// TwinCAT 3 PLC project Samples
// Title: TF8040 PLC-Samples
// Company: Beckhoff Automation GmbH
// Author: Beckhoff Automation
// ProjectVersion: 2.1.1.0
// Description: PLC.Samples to demontrate function volume of TF8040.
// ProgramVersion: 3.1.4023.0
// libraries:
//   Tc2_Standard, * (Beckhoff Automation GmbH)
//   Tc2_System, * (Beckhoff Automation GmbH)
//   Tc2_Utilities, * (Beckhoff Automation GmbH)
//   Tc3_BA2, * (Beckhoff Automation GmbH)
//   Tc3_BA2_Common, * (Beckhoff Automation GmbH)
//   Tc3_BACnetRev14, * (Beckhoff Automation GmbH)
//   Tc3_Module, * (Beckhoff Automation GmbH)
//   Tc3_XBA, * (Beckhoff Automation GmbH)
// project tree:
//   / PlcTask.TcTTO (not stored)
//   SAMPLES/Demo/Event/ FB_Evt_Ack.TcPOU, FB_Evt_EventClasses.TcPOU (not stored), FB_Evt_Events.TcPOU, FB_Evt_Misc.TcPOU, FB_Evt_QueryCnd.TcPOU (not stored)
//   SAMPLES/Demo/Event/Function/ F_AcknowledgeEventClass.TcPOU (not stored)
//   SAMPLES/Demo/Objects/ FB_Obj_AddParam.TcPOU, FB_Obj_General.TcPOU, FB_Obj_Misc.TcPOU, FB_Obj_Sequence.TcPOU (not stored), FB_Obj_UserDefined.TcPOU (not stored)
//   SAMPLES/Demo/Objects/Misc/ E_UDef_Mode.TcDUT (not stored), FB_UDef_BValEx.TcPOU, FB_UDef_SpVal.TcPOU, FB_UDef_SpValEx.TcPOU (not stored)
//   SAMPLES/Demo/Optional Extensions/Events/ FB_MyLocalObjectEvents.TcPOU, FB_MyProjectEvents.TcPOU (not stored)
//   SAMPLES/Demo/Optional Extensions/ MAIN_OPTEXT.TcPOU
//   SAMPLES/Demo/Other/ FB_Misc.TcPOU, FB_Texts.TcPOU (not stored)
//   SAMPLES/Demo/Plant/ FB_Plt_Init1.TcPOU (not stored), FB_Plt_Init2.TcPOU (not stored), FB_Plt_Init3.TcPOU (not stored)
//   SAMPLES/Demo/Reference/ FB_Ref_Collectors.TcPOU (not stored), FB_Ref_Groups.TcPOU (not stored)
//   SAMPLES/Demo/Reference/Publish and Subscribe/ FB_Ref_PubSub_Local.TcPOU (not stored), FB_Ref_PubSub_Remote.TcPOU
//   SAMPLES/Demo/Structure/ FB_Struct_Nested.TcPOU (not stored)
//   SAMPLES/Demo/Supplement specific/BACnet/ FB_BACnet_EvtInh.TcPOU, FB_BACnet_ObjPropRef.TcPOU (not stored), FB_BACnet_RcpList.TcPOU
//   SAMPLES/Demo/Supplement specific/BACnet/Optional Extensions/Events/ FB_BACnet_MyLocalObjectEvents.TcPOU
//   SAMPLES/Demo/Supplement specific/BACnet/Optional Extensions/ MAIN_OPTEXT_BACnet.TcPOU (not stored)
//   SAMPLES/Demo/[Helper]/FunctionBlocks/Aggregates/ FB_TimerAggregateA.TcPOU (not stored), FB_ProcAggregateB.TcPOU (not stored)
//   SAMPLES/Demo/[Helper]/FunctionBlocks/Nested/ FB_NestedView.TcPOU (not stored), FB_NestedView2.TcPOU (not stored), FB_SubNestedView.TcPOU (not stored), FB_SubSubNestedView.TcPOU
//   SAMPLES/ MAIN.TcPOU
//   SAMPLES/Templates/Standard/DUTs/Enumerations/OpMod/ E_OpMod_AC.TcDUT, E_OpMod_Binary.TcDUT (not stored), E_OpMod_ClsOpn.TcDUT (not stored), E_OpMod_Step2.TcDUT (not stored)
//   SAMPLES/Templates/Standard/GVLs/ MyECIDs.TcGVL (not stored), MyLabels.TcGVL (not stored), MyProfiles.TcGVL
//   SAMPLES/Templates/Standard/POUs/Trade/General/Building/ FB_BA_Bld01.TcPOU
//   SAMPLES/Templates/Standard/POUs/Trade/General/EventClasses/ FB_BA_EC01.TcPOU
//   SAMPLES/Templates/User-defined/Objects/ FB_UDef_Obj.TcPOU (not stored)
//   SAMPLES/Templates/User-defined/Sample Weather Station/ FB_BA_MyWeatherStation.TcPOU (not stored), FB_BA_MyWeatherStationSub.TcPOU (not stored), I_BA_MyWeatherStation.TcIO, ST_BA_MyWeatherData.TcDUT
// real-time tasks:
//   TASK PlcTask: cycle T#45ms, priority 20, ADS port 350
//   TASK Device 1 (BACnet IP)_Task_58: cycle T#40ms, priority 58, ADS port 351
//   TASK Gerät 1 (BACnet IP)_QueueTask: cycle T#2ms, priority 8, ADS port 352
// I/O:
//   DEVICE Gerät 1 (BACnet IP), AmsNetId 192.168.216.1.2.1
// variable links:
//   Samples/Samples Instance <-> Device 1 (BACnet IP)
//     PlcTask Inputs/Tc3_BACnetRev14.BACnet_Globals.DefaultAdapter.BACnet_AmsNetId <-> Inputs/AmsNetId

// ---- SAMPLES/Templates/Standard/DUTs/Enumerations/OpMod/E_OpMod_AC.TcDUT
{attribute 'qualified_only'}
TYPE E_OpMod_AC :
(
	Invalid			:= 0,
	
	eOff			:= 1,
	eOn				:= 2,
	eNightCool		:= 3,
	eDisturb		:= 4,
	eSmokeExtract	:= 5,
	eFrost			:= 6,
	eFire			:= 7,
	eCentralOff		:= 8
	
) UDINT;
END_TYPE

// ---- SAMPLES/Templates/User-defined/Sample Weather Station/ST_BA_MyWeatherData.TcDUT
TYPE ST_BA_MyWeatherData :
STRUCT
	fWeatherTemperature		: REAL;
	fHumidity				: REAL;
	fBrightness				: REAL;
	fWindSpeed				: REAL;
	fWindDirection			: REAL;
	fLatitude				: REAL;
	fLongitude				: REAL;
	
	bDisturb				: BOOL;
END_STRUCT
END_TYPE

// ---- SAMPLES/Templates/Standard/GVLs/MyProfiles.TcGVL
{attribute 'qualified_only'}
VAR_GLOBAL
	{region 'Placeholder'}
		{region 'Text'}
			txtOff						: STRING						:= 'Aus';
			txtOn						: STRING						:= 'Ein';
			txtNormal					: STRING						:= 'Normal';
			txtOffnormal				: STRING						:= 'Unnormal';
			txtAlert					: STRING						:= 'Alarm';
			txtDisturb					: STRING						:= 'Störung';
			txtExceeded					: STRING						:= 'Überschritten';
			txtMonitoring				: STRING						:= 'Überwachung';
			txtProtection				: STRING						:= 'Schutzbetrieb';
			txtEconomy					: STRING						:= 'Economy';
			txtComfort					: STRING						:= 'Comfort';
		{endregion}
		{region 'Event Transition Text'}
			trnsExceeded				: T_BA_EventTransitionText		:= [txtExceeded,			txtDisturb,			txtNormal];
			trnsMonitoring				: T_BA_EventTransitionText		:= [txtMonitoring,			txtDisturb,			txtNormal];
		{endregion}
		{region 'Multistate Text'}
			txtEnergyLevel				: T_BA_StateTextArray			:= [txtProtection,			txtEconomy,			txtComfort];
		{endregion}
	{endregion}
END_VAR
VAR_GLOBAL
	{region 'Sample Templates'}
		// A
		// B
		CmdB							: FB_BA_ProfileBEvtObj			:= (sInactiveText := txtOff,			sActiveText := txtOn,			aEventTransitionText := trnsMonitoring,							nEventClassID := 11);
		// D
		// E
		// F
		// G
		// H
		// I
		// J
		// K
		// L
		// M
		// N
		// O
		// P	
		// Q
		// R
		// S	
		// t
		// U
		// v
		// W
		// X
		// Y
		// Z
	{endregion}
	{region 'Sample Objects'}
		{region 'Analog'}
			AV_Prf						: FB_BA_ProfileAEvtObj			:= (eUnit:=E_BA_Unit.eTemperature_DegreesCelsius,						aEventTransitionText:=MyProfiles.trnsExceeded,					nEventClassID:=MyECIDs.AlmStd);
			AVOp_Prf					: FB_BA_ProfileAObj				:= (eUnit:=E_BA_Unit.eTemperature_DegreesCelsius);
			AI_Prf						: FB_BA_ProfileAEvtObj			:= (eUnit:=E_BA_Unit.eTemperature_DegreesCelsius,						aEventTransitionText:=MyProfiles.trnsExceeded,					nEventClassID:=MyECIDs.AlmStd);
			AO_Prf						: FB_BA_ProfileAEvtObj			:= (eUnit:=E_BA_Unit.eTemperature_DegreesCelsius,						aEventTransitionText:=MyProfiles.trnsExceeded,					nEventClassID:=MyECIDs.AlmStd);
		{endregion}
		{region 'Binary'}
			BV_Prf						: FB_BA_ProfileBEvtObj			:= (sInactiveText := txtOff, sActiveText := txtOn,						aEventTransitionText:=MyProfiles.trnsExceeded,					nEventClassID:=MyECIDs.AlmStd);
			BVOp_Prf					: FB_BA_ProfileBObj				:= (sInactiveText := txtOff, sActiveText := txtOn);
			BI_Prf						: FB_BA_ProfileBEvtObj			:= (sInactiveText := txtOff, sActiveText := txtOn,						aEventTransitionText:=MyProfiles.trnsExceeded,					nEventClassID:=MyECIDs.AlmStd);
			BO_Prf						: FB_BA_ProfileBEvtObj			:= (sInactiveText := txtOff, sActiveText := txtOn,						aEventTransitionText:=MyProfiles.trnsExceeded,					nEventClassID:=MyECIDs.AlmStd);
		{endregion}
		{region 'Multistate'}
			MV_Prf						: FB_BA_ProfileMEvtObj			:= (aStateText:=MyProfiles.txtEnergyLevel,								aEventTransitionText:=MyProfiles.trnsExceeded,					nEventClassID:=MyECIDs.AlmStd);	
			MVOp_Prf					: FB_BA_ProfileMObj				:= (aStateText:=MyProfiles.txtEnergyLevel);
			MI_Prf						: FB_BA_ProfileMEvtObj			:= (aStateText:=MyProfiles.txtEnergyLevel,								aEventTransitionText:=MyProfiles.trnsExceeded,					nEventClassID:=MyECIDs.AlmStd);
			MO_Prf						: FB_BA_ProfileMEvtObj			:= (aStateText:=MyProfiles.txtEnergyLevel,								aEventTransitionText:=MyProfiles.trnsExceeded,					nEventClassID:=MyECIDs.AlmStd);
		{endregion}
		{region 'Misc'}
			Loop_Prf					: FB_BA_ProfileAObj				:= (eUnit:=E_BA_Unit.eOther_Percent);
			Cal_Prf						: FB_BA_ProfileBObj				:= (sInactiveText := txtOff, sActiveText := txtOn);
			SchedA_Prf					: FB_BA_ProfileAObj				:= (eUnit:=E_BA_Unit.eOther_Percent);
			SchedB_Prf					: FB_BA_ProfileBObj				:= (sInactiveText := txtOff, sActiveText := txtOn);
			SchedM_Prf					: FB_BA_ProfileMObj				:= (aStateText:=MyProfiles.txtEnergyLevel);
			Trend_Prf					: FB_BA_ProfileBObj				:= (sInactiveText := txtOff, sActiveText := txtOn);
			EvtCls_Prf					: FB_BA_Profile;
		{endregion}
		{region 'Custom'}
			MyWthSt_Prf					: FB_BA_Profile;
		{endregion}
		{region 'Collectors'}
			Col_PrfEn					: FB_BA_ProfileBObj				:= (sInactiveText := 'Nein', sActiveText := 'Ja');
			Col_PrfValA					: FB_BA_ProfileAObj				:= (eUnit:=E_BA_Unit.eTemperature_DegreesCelsius);
		{endregion}
	{endregion}
END_VAR

// ---- SAMPLES/Templates/User-defined/Sample Weather Station/I_BA_MyWeatherStation.TcIO
INTERFACE I_BA_MyWeatherStation EXTENDS I_BA_Publisher

PROPERTY Brightness : REAL
GET
END_GET
END_PROPERTY

PROPERTY Error : BOOL
GET
END_GET
END_PROPERTY

PROPERTY Humidity : REAL
GET
END_GET
END_PROPERTY

PROPERTY Latitude : REAL
GET
END_GET
END_PROPERTY

PROPERTY Longitude : REAL
GET
END_GET
END_PROPERTY

PROPERTY Ready : BOOL
GET
END_GET
END_PROPERTY

PROPERTY WeatherTemperature : REAL
GET
END_GET
END_PROPERTY

PROPERTY WindDirection : REAL
GET
END_GET
END_PROPERTY

PROPERTY WindSpeed : REAL
GET
END_GET
END_PROPERTY

END_INTERFACE

// ---- SAMPLES/Demo/Event/FB_Evt_Ack.TcPOU
// Acknowledgement-Examples.
// > One object per demonstrated 'AlarmMode'.
// > See "FB_BA_EC01" to view decleared event classes.
// [Hint]
// > All reference-variables are implemented to ease monitoring of relevant variables.
// > show the possibility to acknowledge BA objects assigned to a specific event class.
FUNCTION_BLOCK FB_Evt_Ack EXTENDS FB_BA_View
VAR               
	{region 'General'}
		bAlm_Test						: BOOL;																						// Trigger alarm for testing.
		bAlm_AckAll						: REFERENCE TO BOOL							REF= THIS^.bAcknowledgeRm;						// Acknowledge all test objects.
		bAlm_AckMode					: POINTER TO BOOL							:= ADR(XBA_Param.eEvtMgmt_AckMode);				// Used reset mode (See parameter description for more details)
	{endregion}
		 
	{region 'Simple'}
		// Intention:					Alarm that automatically disappears.
		// State on active alarm:		- "bEvent = TRUE'
		//								- "stAckedTransitions = [FALSE,true,true]'
		// State when disappeared:		- "bEvent = false'
		//								- "stAckedTransitions = [true,true,true]'
		AlmSimple_Ack					: REFERENCE TO BOOL							REF= AlmSimple.bAcknowledgeRm;
		AlmSimple_Indicated				: BOOL;
		AlmSimple_Event					: REFERENCE TO BOOL							REF= AlmSimple.bEvent;
		AlmSimple						: FB_BA_BI_Raw := (
											iParent									:= THIS^,
											sInactiveText							:= 'Normal',
											sActiveText								:= 'Alarm',
											nEventClassID							:= MyECIDs.AlmSmpl);
	{endregion}
	{region 'Standard'}
		// Intention:					Alarm that is just indicated (by acknowledge transition) when disappeared.
		// State on active alarm:		- "bEvent = TRUE'
		//								- "stAckedTransitions = [FALSE,true,true]'
		// State when disappeared:		- "bEvent = false'
		//								- "stAckedTransitions = [FALSE,true,true]'
		// State after acknowledgement:	- "bEvent = false'
		//								- "stAckedTransitions = [true,true,true]'
		AlmStandard_Ack					: REFERENCE TO BOOL							REF= AlmStandard.bAcknowledgeRm;
		AlmStandard_Indicated			: BOOL;
		AlmStandard_Event				: REFERENCE TO BOOL							REF= AlmStandard.bEvent;
		AlmStandard						: FB_BA_BI_Raw := (
											iParent									:= THIS^,
											sInactiveText							:= 'Normal',
											sActiveText								:= 'Alarm',
											nEventClassID							:= MyECIDs.AlmStd);	
	{endregion}
	{region 'Extended'}
		// Intention:					Alarm that is indicated (by acknowledge transition) and hold when disappeared.
		//								The 'bEvent' is released when an additional reset has been triggered.
		// State on active alarm:		- "bEvent = TRUE'
		//								- "stAckedTransitions = [FALSE,true,FALSE]'
		// State when disappeared:		- "bEvent = TRUE'
		//								- "stAckedTransitions = [FALSE,true,FALSE]'
		// State after acknowledgement:	- "bEvent = TRUE'
		//								- "stAckedTransitions = [true,true,FALSE]'
		// State after reset:			- "bEvent = false'
		//								- "stAckedTransitions = [true,true,true]'
		AlmExtended_Ack					: REFERENCE TO BOOL							REF= AlmExtended.bAcknowledgeRm;
		AlmExtended_Indicated			: BOOL;
		AlmExtended_Event				: REFERENCE TO BOOL							REF= AlmExtended.bEvent;
		AlmExtended						: FB_BA_BI_Raw := (
											iParent									:= THIS^,
											sInactiveText							:= 'Normal',
											sActiveText								:= 'Alarm',
											nEventClassID							:= MyECIDs.AlmExt);	
	{endregion}	
		 
	{region 'Acknowledge event class'}	
		// Intention:					Acknowledge all objects that reference a specific event class.
		nEventClassID					: UINT										:= 0;			// Enter ID of event class to acknowledge.
	{endregion}
		 
END_VAR

SUPER^();

AlmSimple(bRawVal:=bAlm_Test);
AlmSimple_Indicated := (NOT AlmSimple.stAckedTransitions.bToOffnormal);
AlmStandard(bRawVal:=bAlm_Test);
AlmStandard_Indicated := (NOT AlmStandard.stAckedTransitions.bToOffnormal);
AlmExtended(bRawVal:=bAlm_Test);
AlmExtended_Indicated := (NOT AlmExtended.stAckedTransitions.bToOffnormal);

IF (nEventClassID <> 0) THEN
	F_AcknowledgeEventClass(nEventClassID);
	nEventClassID := 0;
END_IF

// Intention:			Illustrate how to recognize changed events.
METHOD PROTECTED OnObjectEventChange
VAR_INPUT
	iObject				: I_BA_EventObject;
	bNotifyParents		: BOOL				:= TRUE;
END_VAR
SUPER^.OnObjectEventChange(iObject, bNotifyParents);

// Sample 1) Evaluate current event state:
CASE (iObject.EventIcon.eState) OF
	E_BA_EventIconState.eGoneAcked,
	E_BA_EventIconState.ePresentAcked:
		iObject.LogMsg.Show(ADSLOG_MSGTYPE_HINT, 'OOEC06', 'Object acknowledged.', TRUE);
END_CASE

// Sample 2) Compare actual event state to previous event state:
IF (iObject.LastEventIcon.eState < iObject.EventIcon.eState) THEN
	; // State intensed...
ELSE
	; // State softened...
END_IF
END_METHOD

END_FUNCTION_BLOCK

// ---- SAMPLES/Demo/Event/FB_Evt_Events.TcPOU
// Examples of objects that refer different event classes.
// > One object per 'EventType' and 'AlarmMode'.
// > One "PlantLock" per 'EventType'.
// > One "PlantLock" for entire view.
// > See "FB_BA_EC01" to view decleared event classes.
// [Hint]
// > All reference-variables are implemented to ease monitoring of relevant variables.
FUNCTION_BLOCK FB_Evt_Events EXTENDS FB_BA_View
VAR
	{region 'General'}
		Lock					: FB_BA_PlantLock				:= (iParent:=THIS^);
	{endregion}
		 
	{region 'Alarm'}
		Alm						: FB_BA_View					:= (iParent:=THIS^,	sDescription:='{Alarm}');
			AlmLock				: FB_BA_PlantLock				:= (iParent:=Alm);
							
			BIAlmSmpl_Val		: REFERENCE TO BOOL				REF= BIAlmSmpl.bVal;
			BIAlmSmpl_LockPrio	: POINTER TO E_BA_LockPriority	:= ADR(BIAlmSmpl.eEnPlantLock);
			BIAlmSmpl			: FB_BA_BI						:= (iParent:=Alm,	iLabel:=MyLabels.Cmd,	iProfile:=MyProfiles.CmdB,	nEventClassID:=MyECIDs.AlmSmpl);
			BIAlmStd_Val		: REFERENCE TO BOOL				REF= BIAlmStd.bVal;
			BIAlmStd_LockPrio	: POINTER TO E_BA_LockPriority	:= ADR(BIAlmStd.eEnPlantLock);
			BIAlmStd			: FB_BA_BI						:= (iParent:=Alm,	iLabel:=MyLabels.Cmd,	iProfile:=MyProfiles.CmdB,	nEventClassID:=MyECIDs.AlmStd,	eEnPlantLock:= E_BA_LockPriority.eHigh);
			BIAlmExt_Val		: REFERENCE TO BOOL				REF= BIAlmExt.bVal;
			BIAlmExt_LockPrio	: POINTER TO E_BA_LockPriority	:= ADR(BIAlmExt.eEnPlantLock);
			BIAlmExt			: FB_BA_BI						:= (iParent:=Alm,	iLabel:=MyLabels.Cmd,	iProfile:=MyProfiles.CmdB,	nEventClassID:=MyECIDs.AlmExt);
	{endregion}
	{region 'Disturb'}
		Dstb					: FB_BA_View					:= (iParent:=THIS^,	sDescription:='{Disturb}');
			DstbLock			: FB_BA_PlantLock				:= (iParent:=Dstb);

			BIDstbSmpl_Val		: REFERENCE TO BOOL				REF= BIDstbSmpl.bVal;
			BIDstbSmpl_LockPrio	: POINTER TO E_BA_LockPriority	:= ADR(BIDstbSmpl.eEnPlantLock);
			BIDstbSmpl			: FB_BA_BI						:= (iParent:=Dstb,	iLabel:=MyLabels.Cmd,	iProfile:=MyProfiles.CmdB,	nEventClassID:=MyECIDs.DstSmpl);
			BIDstbStd_Val		: REFERENCE TO BOOL				REF= BIDstbStd.bVal;
			BIDstbStd_LockPrio	: POINTER TO E_BA_LockPriority	:= ADR(BIDstbStd.eEnPlantLock);
			BIDstbStd			: FB_BA_BI						:= (iParent:=Dstb,	iLabel:=MyLabels.Cmd,	iProfile:=MyProfiles.CmdB,	nEventClassID:=MyECIDs.DstStd,	eEnPlantLock:= E_BA_LockPriority.eMedium);
			BIDstbExt_Val		: REFERENCE TO BOOL				REF= BIDstbExt.bVal;
			BIDstbExt_LockPrio	: POINTER TO E_BA_LockPriority	:= ADR(BIDstbExt.eEnPlantLock);
			BIDstbExt			: FB_BA_BI						:= (iParent:=Dstb,	iLabel:=MyLabels.Cmd,	iProfile:=MyProfiles.CmdB,	nEventClassID:=MyECIDs.DstExt);
	{endregion}
	{region 'Maintenance'}
		Mntn					: FB_BA_View					:= (iParent:=THIS^,	sDescription:='{Maintenance}');
			MntnLock			: FB_BA_PlantLock				:= (iParent:=Mntn);

			BIMntnSmpl_Val		: REFERENCE TO BOOL				REF= BIMntnSmpl.bVal;
			BIMntnSmpl_LockPrio	: POINTER TO E_BA_LockPriority	:= ADR(BIMntnSmpl.eEnPlantLock);
			BIMntnSmpl			: FB_BA_BI						:= (iParent:=Mntn,	iLabel:=MyLabels.Cmd,	iProfile:=MyProfiles.CmdB,	nEventClassID:=MyECIDs.MntnSmpl);
			BIMntnStd_Val		: REFERENCE TO BOOL				REF= BIMntnStd.bVal;
			BIMntnStd_LockPrio	: POINTER TO E_BA_LockPriority	:= ADR(BIMntnStd.eEnPlantLock);
			BIMntnStd			: FB_BA_BI						:= (iParent:=Mntn,	iLabel:=MyLabels.Cmd,	iProfile:=MyProfiles.CmdB,	nEventClassID:=MyECIDs.MntnStd,	eEnPlantLock:= E_BA_LockPriority.eLocalHigh);
			BIMntnExt_Val		: REFERENCE TO BOOL				REF= BIMntnExt.bVal;
			BIMntnExt_LockPrio	: POINTER TO E_BA_LockPriority	:= ADR(BIMntnExt.eEnPlantLock);
			BIMntnExt			: FB_BA_BI						:= (iParent:=Mntn,	iLabel:=MyLabels.Cmd,	iProfile:=MyProfiles.CmdB,	nEventClassID:=MyECIDs.MntnExt);
	{endregion}
	{region 'Notification'}
		Ntfy					: FB_BA_View					:= (iParent:=THIS^,	sDescription:='{Notification}');
			NtfyLock			: FB_BA_PlantLock				:= (iParent:=Ntfy);

			BINtfySmpl_Val		: REFERENCE TO BOOL				REF= BINtfySmpl.bVal;
			BINtfySmpl_LockPrio	: POINTER TO E_BA_LockPriority	:= ADR(BINtfySmpl.eEnPlantLock);
			BINtfySmpl			: FB_BA_BI						:= (iParent:=Ntfy,	iLabel:=MyLabels.Cmd,	iProfile:=MyProfiles.CmdB,	nEventClassID:=MyECIDs.NtfSmpl);
			BINtfyStd_Val		: REFERENCE TO BOOL				REF= BINtfyStd.bVal;
			BINtfyStd_LockPrio	: POINTER TO E_BA_LockPriority	:= ADR(BINtfyStd.eEnPlantLock);
			BINtfyStd			: FB_BA_BI						:= (iParent:=Ntfy,	iLabel:=MyLabels.Cmd,	iProfile:=MyProfiles.CmdB,	nEventClassID:=MyECIDs.NtfStd,	eEnPlantLock:= E_BA_LockPriority.eLocalMedium);
	{endregion}
	{region 'Other'}
		Other					: FB_BA_View					:= (iParent:=THIS^,	sDescription:='{Other}');
			OtherLock			: FB_BA_PlantLock				:= (iParent:=Other);
				 
			BIOthrSmpl_Val		: REFERENCE TO BOOL				REF= BIOthrSmpl.bVal;
			BIOthrSmpl_LockPrio	: POINTER TO E_BA_LockPriority	:= ADR(BIOthrSmpl.eEnPlantLock);
			BIOthrSmpl			: FB_BA_BI						:= (iParent:=Other,	iLabel:=MyLabels.Cmd,	iProfile:=MyProfiles.CmdB,	nEventClassID:=MyECIDs.OthSmpl);
			BIOthrStd_Val		: REFERENCE TO BOOL				REF= BIOthrStd.bVal;
			BIOthrStd_LockPrio	: POINTER TO E_BA_LockPriority	:= ADR(BIOthrStd.eEnPlantLock);
			BIOthrStd			: FB_BA_BI						:= (iParent:=Other,	iLabel:=MyLabels.Cmd,	iProfile:=MyProfiles.CmdB,	nEventClassID:=MyECIDs.OthStd);
	{endregion}                                                
END_VAR

SUPER^(); // FB_BA_View
Lock(); // FB_BA_PlantLock
Alm(); // FB_BA_View
AlmLock(); // FB_BA_PlantLock
BIAlmSmpl(); // FB_BA_BI
BIAlmStd(); // FB_BA_BI
BIAlmExt(); // FB_BA_BI
Dstb(); // FB_BA_View
DstbLock(); // FB_BA_PlantLock
BIDstbSmpl(); // FB_BA_BI
BIDstbStd(); // FB_BA_BI
BIDstbExt(); // FB_BA_BI
Mntn(); // FB_BA_View
MntnLock(); // FB_BA_PlantLock
BIMntnSmpl(); // FB_BA_BI
BIMntnStd(); // FB_BA_BI
BIMntnExt(); // FB_BA_BI
Ntfy(); // FB_BA_View
NtfyLock(); // FB_BA_PlantLock
BINtfySmpl(); // FB_BA_BI
BINtfyStd(); // FB_BA_BI
Other(); // FB_BA_View
OtherLock(); // FB_BA_PlantLock
BIOthrSmpl(); // FB_BA_BI
BIOthrStd(); // FB_BA_BI

END_FUNCTION_BLOCK

// ---- SAMPLES/Demo/Event/FB_Evt_Misc.TcPOU
FUNCTION_BLOCK FB_Evt_Misc EXTENDS FB_BA_View
VAR
	{region 'Iteration'}
		// Intention:			Iterate over active events.
		bIterate				: BOOL;
		bIterate_ShowTimestamp	: BOOL				:= FALSE;
		bIterate_ShowType		: BOOL				:= TRUE;
		bIterate_ShowState		: BOOL				:= TRUE;
		bIterate_ShowEC			: BOOL				:= FALSE;
	{endregion}
END_VAR
VAR
	_i							: DINT;
	_sVal						: T_MaxString;
	_iObj						: I_BA_EventObject;
	_fbMsg						: FB_BA_DecorString;
END_VAR

SUPER^();

IF (bIterate) THEN
	bIterate := FALSE;
	
	_i := F_BA_GetEventCount();
	IF (_i = 0) THEN
		F_BA_LogMessage(ADSLOG_MSGTYPE_HINT, 'EM06', 'No active events found yet.');
	ELSE
		F_BA_LogMessage1(ADSLOG_MSGTYPE_HINT, 'EM08', 'Active events: %d', F_DINT(_i));
		
		// Iterate over all active events:
		_i := 0;
		_iObj := 0;								// [Hint] Temporary iterator-object must be NULL to start iteration from the beginning.
		WHILE (F_BA_IterateEvents(_iObj)) DO
			_i := (_i+1);
			
			// Format message:
			_fbMsg.Reset();
			IF (bIterate_ShowTimestamp) THEN
				_sVal := TO_STRING(F_BA_ToDT(_iObj.EventChangeTime));
				_fbMsg.AddDecor1('%s', F_STRING(_sVal));
			END_IF
			IF (bIterate_ShowType) THEN
				_fbMsg.AddDecor1('Type: %s', F_STRINGEx(BA_EnumEN.aEventType[_iObj.EventIcon.eEventType].sName));
			END_IF
			IF (bIterate_ShowState) THEN
				_fbMsg.AddDecor1('State: %s', F_STRINGEx(BA_EnumEN.aEventIconState[_iObj.EventIcon.eState].sDescription));
			END_IF
			IF (bIterate_ShowEC) THEN
				_sVal := TO_STRING(_iObj.EventClassID);
				_fbMsg.AddDecor1('Event class: %s', F_STRING(_sVal));
			END_IF
			_fbMsg.Finish();
			
			_sVal := _iObj.ObjectName;
			F_BA_LogMessage3(ADSLOG_MSGTYPE_HINT, 'EM32', '%d. %s   %s', F_DINT(_i), F_STRING(_sVal), F_STRING(_fbMsg.sOutput));
		END_WHILE
	END_IF
END_IF

END_FUNCTION_BLOCK

// ---- SAMPLES/Demo/Objects/FB_Obj_AddParam.TcPOU
FUNCTION_BLOCK FB_Obj_AddParam EXTENDS FB_BA_View
VAR
	TestSpVal			: FB_UDef_SpVal := (
							iParent					:= THIS^,		
							sDescription			:= 'My user defined setpoint object',
							eMode					:= E_UDef_Mode.eAdd
						);
	TestSpValEx			: FB_UDef_SpValEx := (
							iParent					:= THIS^,
							sDescription			:= 'Another user defined enabled setpoint object',
							eMode					:= E_UDef_Mode.eSubstract
						);
	TestBValEx			: FB_UDef_BValEx := (
							iParent					:= THIS^,
							sDescription			:= 'My user defined boolean value extension',
							sActiveText				:= 'Active',
							sInactiveText			:= 'Inactive'
						);
END_VAR
VAR
	{region 'Test'}
		nOffset			: UINT						:= 3;
	{endregion}
END_VAR

SUPER^(); // FB_BA_View
TestSpVal(nSomeOffset := nOffset); // FB_UDef_SpVal
TestSpValEx(nSomeOffset := nOffset); // FB_UDef_SpValEx
TestBValEx(); // FB_UDef_BValEx

END_FUNCTION_BLOCK

// ---- SAMPLES/Demo/Objects/Misc/FB_UDef_SpVal.TcPOU
// User defined setpoint providing value.
// > Contains additional parameters.
FUNCTION_BLOCK FB_UDef_SpVal EXTENDS FB_BA_Object
VAR_INPUT CONSTANT
	{region 'Variable Parameters'}
		{attribute 'BaParam.Title.DE' := 'Irgendein Sollwert'}
		{attribute 'BaParam.Title.EN' := 'Some setpoint'}
		{attribute 'BaParam.Access.Read' := 'Guest'}
		{attribute 'BaParam.Access.Write' := 'Basic'}
		fSomeSetpoint : REAL := 10.0;
	{endregion}
END_VAR
VAR_INPUT
	{attribute 'BaParam.Title.DE' := 'Irgendein Offset'}
	{attribute 'BaParam.Title.EN' := 'Some offset'}
	{attribute 'BaParam.Access.Read' := 'Guest'}
	nSomeOffset : UINT := 3;
END_VAR
VAR_OUTPUT
	{attribute 'BaParam.Title.DE' := 'Ergebnis'}
	{attribute 'BaParam.Title.EN' := 'Result'}
	{attribute 'BaParam.Access.Read' := 'Guest'}
	fResult : REAL;
END_VAR
VAR
	{attribute 'BaParam.Title.DE' := 'Modus'}
	{attribute 'BaParam.Title.EN' := 'Mode'}
	{attribute 'BaParam.Access.Read' := 'Advanced'}
	{attribute 'BaParam.Access.Write' := 'Expert'}
	eMode : E_UDef_Mode := E_UDef_Mode.eAdd;
END_VAR

SUPER^();

CASE (eMode) OF
	E_UDef_Mode.eAdd: fResult := (fSomeSetpoint + TO_REAL(nSomeOffset));
	E_UDef_Mode.eSubstract: fResult := (fSomeSetpoint - TO_REAL(nSomeOffset));
ELSE
	fResult := fSomeSetpoint;
END_CASE

END_FUNCTION_BLOCK

// ---- SAMPLES/Demo/Objects/Misc/FB_UDef_BValEx.TcPOU
// User defined boolean value extension.
// > Contains additional parameters.
FUNCTION_BLOCK FB_UDef_BValEx EXTENDS FB_BA_BV_OP
VAR_INPUT CONSTANT
	{region 'Variable Parameters'}
		{attribute 'BaParam.Title.DE' := 'Erwarteter Wert'}
		{attribute 'BaParam.Title.EN' := 'Expected value'}
		{attribute 'BaParam.Access.Read' := 'Guest'}
		{attribute 'BaParam.Access.Write' := 'Advanced'}
		bExpected : BOOL;
	{endregion}
END_VAR
VAR_OUTPUT
	{attribute 'BaParam.Title.DE' := 'Übereinstimmend'}
	{attribute 'BaParam.Title.EN' := 'Matched'}
	{attribute 'BaParam.Access.Read' := 'Guest'}
	bMatch : BOOL;
END_VAR

SUPER^();

bMatch := (bPresentValue = bExpected);

END_FUNCTION_BLOCK

// ---- SAMPLES/Demo/Optional Extensions/Events/FB_MyLocalObjectEvents.TcPOU
FUNCTION_BLOCK FB_MyLocalObjectEvents EXTENDS FB_BA_LocalObjectEventSubscriber

METHOD PRIVATE IsPressure : BOOL
VAR_INPUT
	eUnit		: E_BA_Unit;
END_VAR
IsPressure := (E_BA_Unit.ePressure_Pascals <= eUnit) AND_THEN (eUnit <= E_BA_Unit.ePressure_InchesOfMercury);
END_METHOD

METHOD PRIVATE IsTemperature : BOOL
VAR_INPUT
	eUnit		: E_BA_Unit;
END_VAR
IsTemperature := (E_BA_Unit.eTemperature_DegreesCelsius <= eUnit) AND_THEN (eUnit <= E_BA_Unit.eTemperature_DegreeDaysFahrenheit);
END_METHOD

METHOD PROTECTED OnInitInstanceId
VAR_INPUT
	iObject			: I_BA_Object;
END_VAR
VAR_INST
	_nID_Temp		: UDINT						:= 5000;				// First ID to assign to temperature sensors.
	_nID_Prs		: UDINT						:= 6000;				// First ID to assign to pressure sensors.
END_VAR
VAR
	_iAnalogObj		: I_BA_AnalogObject;
	_nID			: REFERENCE TO UDINT;
END_VAR
// Sample 1) Generate instance ID related to configured units.

IF (iObject.InstanceID <> 0) THEN
	; // ID already assigned.
ELSIF (iObject.DataClass <> E_BA_DataClass.eAnalog) THEN
	; // Skip.
ELSIF (NOT __QUERYINTERFACE(iObject, _iAnalogObj)) THEN
	; // Failed to convert interface.
ELSE
	// Determine range of instance IDs:
	IF (IsTemperature(_iAnalogObj.Unit)) THEN
		_nID REF= _nID_Temp;
	ELSIF (IsPressure(_iAnalogObj.Unit)) THEN
		_nID REF= _nID_Prs;
	ELSE
		RETURN; // Skip (Instance ID will be auto-generated).
	END_IF
		
	// Assign instance ID:
	_iAnalogObj.InstanceID := _nID;
	iObject.LogMsg.Show1(ADSLOG_MSGTYPE_HINT, 'OIII21', 'Assigned instance ID %d.', F_UDINT(_nID), FALSE);
	
	_nID := (_nID+1);
END_IF
END_METHOD

END_FUNCTION_BLOCK

// ---- SAMPLES/Demo/Optional Extensions/MAIN_OPTEXT.TcPOU
// Optional extensions.
// [Hint]
// - To stay maintainable and sustain a nice project overview it is recommended to declare these tools in your MAIN program.
PROGRAM MAIN_OPTEXT
VAR
	{region 'Settings'}
		// Intention:		Adjust certain ("BA_Param" related) settings via PLC code.
		//					> Feel free to implement as much instances as needed, where ever needed.
		Parameters			: FB_BA_Param := (
								EventEn_Simple			:= F_BA_EventTransition(TRUE, FALSE, FALSE),
								EventEn_Standard		:= F_BA_EventTransition(TRUE, FALSE, FALSE),
								EventEn_Extended		:= F_BA_EventTransition(TRUE, FALSE, TRUE),
								EvtMgmt_AckMode			:= E_BA_AcknowledgeMode.eSingle,
								
								// Intention:			Adjust access to some specific parameters (Leaving rest untouched).
								DefWriteAccess			:= F_BA_ParameterRolesBuilder()
															.Set(E_BA_Parameter.eEventEnable, E_BA_Role.eInternal)
															.Build()
							);

		// Intention:		Generically subscribe to certain events.
		//					> Use carefully (Refer to documentation - event subscribers are powerfull!)
		Events_Proj			: FB_MyProjectEvents;
		Events_LocObj		: FB_MyLocalObjectEvents;
	{endregion}
END_VAR

END_PROGRAM

// ---- SAMPLES/Demo/Other/FB_Misc.TcPOU
// Miscellaneous.
FUNCTION_BLOCK FB_Misc EXTENDS FB_BA_View
VAR	
	// Intention:		Take care of UTF-8 encoding manually.
	//					> [Hint] Disable the integrated encoding mechanism (See "BA_Param.bUtf8AutoConvert")!
	SpecialUtf8			: FB_BA_AV_Op := (
							iParent					:= THIS^,
							sDescription			:= wsLiteral_TO_UTF8("{äöüßéèêµ€° Ἀθῆναι İstanbul Київ}"),
							eUnit					:= E_BA_Unit.eOther_Percent,
							fValueRm				:= 5
						);
END_VAR

SUPER^();

SpecialUtf8();

END_FUNCTION_BLOCK

// ---- SAMPLES/Demo/Objects/FB_Obj_General.TcPOU
// Demonstration of objects.
// > See "FB_BA_EC01" to view decleared event classes.
FUNCTION_BLOCK FB_Obj_General EXTENDS FB_BA_View
VAR
	{region 'Analog'}
		A										: FB_BA_View := (
													iParent									:= THIS^,
													sDescription							:= '{Analog objects}'
												);
			 
			// Intention:						Value
			AV									: FB_BA_AV := (
													iParent									:= A,
													sDescription							:= '{Analog Value}',
													eUnit									:= E_BA_Unit.eOther_Percent,
													nEventClassID							:= MyECIDs.AlmStd,
													stLowLimit								:= F_BA_Limit(TRUE, 0),
													stHighLimit								:= F_BA_Limit(TRUE, 50),
													stTimeDelay								:= F_BA_TimeDelay(1, 1),
													bEnPgm									:= TRUE,
													fValPgm									:= 10.0
												);
													
			// Intention:						Value for Display
			// Operation:						Display
			fAVDsp_ValuePgm						: REAL := 0;
			AVDsp								: FB_BA_AV_Op := (
													iParent									:= A,
													sObjectName								:= '{MyAvDsp}',
													sDescription							:= '{Sample AV Display}',
													eUnit									:= E_BA_Unit.eOther_Percent
												);	
			
			// Intention:						Value for Setpoint
			// Operation:						Setpoint
			AVSp								: FB_BA_AV_Op := (
													iParent									:= A,
													sDescription							:= '{Sample AV Setpoint}',
													eUnit									:= E_BA_Unit.eTemperature_DegreesCelsius,
													fValueRm								:= 3
												);
			bAVSp2_ValViaProp					: BOOL;
			fAVSp2_ValViaProp					: REAL;
			AVSp2								: FB_BA_AV_Op := (
													iParent									:= A,
													sDescription							:= '{Sample AV Setpoint 2}',
													eUnit									:= E_BA_Unit.eTemperature_DegreesCelsius,
													fValueRm								:= 3
												);
		
			// Intention:						Input
			// Hardware:						Process Data
			fAI_Proc_ValuePgm					: REAL := 20;
			AI_Proc								: FB_BA_AI := (
													iParent									:= A,
													sDescription							:= '{Sample AI (Process Data)}',
													sDeviceType								:= 'Analoger Eingang',
													eUnit									:= E_BA_Unit.eOther_Percent,
													nEventClassID							:= MyECIDs.AlmStd
												);
		
			// Intention:						Input
			// Hardware:						Raw Data
			AI_Raw								: FB_BA_AI_Raw := (
													iParent									:= A,
													sDescription							:= '{Sample AI (Raw)}',
													sDeviceType								:= 'Analoger Eingang',
													eUnit									:= E_BA_Unit.eOther_Percent,
													nEventClassID							:= MyECIDs.AlmStd
												);
		
			// Intention:						Input
			// Hardware:						I/O
			AI_IO								: FB_BA_AI_IO := (
													iParent									:= A,
													sDescription							:= '{Sample AI (IO)}',
													sDeviceType								:= 'Analoger Eingang',
													eUnit									:= E_BA_Unit.eOther_Percent,
													nEventClassID							:= MyECIDs.AlmStd
												);
												
			AI_IO_2_10V							: FB_BA_AI_IO := (
													iParent									:= A,
													sDescription							:= '{Sample AI (IO)}',
													sDeviceType								:= 'Analoger Eingang (2-10V)',
													eUnit									:= E_BA_Unit.eOther_Percent,
													nEventClassID							:= MyECIDs.AlmStd
												);
		
			// Intention:						Input
			// Hardware:						I/O
			AI_Temp								: FB_BA_AI_IOEx := (
													iParent									:= A,
													sDescription							:= '{Sample AI Temperaturfühler (Temp)}',
													sDeviceType								:= 'Temperaturfühler',
													eUnit									:= E_BA_Unit.eTemperature_DegreesCelsius,
													eSensor									:= E_BA_MeasuringElement.eNI1000,
													nEventClassID							:= MyECIDs.AlmStd
												);
		
			// Intention:						Input for Display
			// Operation:						Display
			// Hardware:						I/O
			// Parameter:						EventDetectionEnable = FALSE
			AIDsp_IO							: FB_BA_AI_IO := (
													iParent									:= A,
													sDescription							:= '{Sample AI Display (IO)}',
													sDeviceType								:= 'Analoger Eingang',
													eUnit									:= E_BA_Unit.eOther_Percent,
													bEventDetectionEnable					:= FALSE,
													nEventClassID							:= MyECIDs.AlmStd
												);
		
			// Intention:						Output
			// Hardware:						Process Data
			AO_CmdProc							: FB_BA_AO := (
													iParent									:= A,
													sDescription							:= '{Analog Befehl (Process Data)}',
													eUnit									:= E_BA_Unit.eOther_Percent,
													nEventClassID							:= MyECIDs.AlmStd
												);
		
			// Intention:						Output
			// Hardware:						Raw Data
			AO_CmdRaw							: FB_BA_AO_Raw := (
													iParent									:= A,
													sDescription							:= '{Analog Befehl (Raw Data)}',
													eUnit									:= E_BA_Unit.eOther_Percent,
													nEventClassID							:= MyECIDs.AlmStd
												);
		
			// Intention:						Output
			// Hardware:						I/O
			AO_CmdIO							: FB_BA_AO_IO := (
													iParent									:= A,
													sDescription							:= '{Analog Befehl (IO)}',
													eUnit									:= E_BA_Unit.eOther_Percent,
													nEventClassID							:= MyECIDs.AlmStd
												);
		
			// Intention:						Output for Display
			// Operation:						Display
			// Hardware:						I/O
			// Parameter:						EventDetectionEnable = FALSE
			AODisp_CmdIO						: FB_BA_AO_IO := (
													iParent									:= A,
													sDescription							:= '{Analog Befehl Display (IO)}',
													eUnit									:= E_BA_Unit.eOther_Percent,
													bEventDetectionEnable					:= FALSE,
													nEventClassID							:= MyECIDs.AlmStd
												);
	{endregion}
	{region 'Binary'}
		B										: FB_BA_View := (
													iParent									:= THIS^,
													sDescription							:= '{Binary objects}'
												);
			 
			// Intention:						Value
			BV									: FB_BA_BV := (
													iParent									:= B,
													sDescription							:= '{Binary Value}',
													sInactiveText							:= 'Aus',
													sActiveText								:= 'Ein',
													nEventClassID							:= MyECIDs.AlmExt
												);
															
			// Intention:						Value for Display
			// Operation:						Display
			bBVDsp_ValuePgm						: BOOL := FALSE;
			BVDsp								: FB_BA_BV_Op := (
													iParent									:= B,
													sDescription							:= '{Sample BV Display}',
													sInactiveText							:= 'Aus',
													sActiveText								:= 'Ein'
												);
			
			// Intention:						Value for Setpoint
			// Operation:						Setpoint
			BVSp								: FB_BA_BV_Op := (
													iParent									:= B,
													sDescription							:= '{Sample BV Setpoint}',
													sInactiveText							:= 'Aus',
													sActiveText								:= 'Ein',
													bValueRm								:= TRUE
												);
												
			// Intention:						Value for Setpoint
			// Operation:						Pushbutton
			nBVPushButton_Counter				: UINT;
			BVPushButton						: FB_BA_BV_Op := (
													iParent									:= B,
													sDescription							:= '{Sample BV Pushbutton}',
													sInactiveText							:= 'Aus',
													sActiveText								:= 'Ein',
													eToggleMode								:= E_BA_ToggleMode.ePushButton
												);
		
			// Intention:						Input
			// Hardware:						Process Data
			BI_Proc								: FB_BA_BI := (
													iParent									:= B,
													sDescription							:= '{Sample BI (Process Data)}',
													sDeviceType								:= 'Sicherung',
													sInactiveText							:= 'Normal',
													sActiveText								:= 'Ausgelöst',
													nEventClassID							:= MyECIDs.AlmStd
												);
		
			// Intention:						Input
			// Hardware:						Raw Data
			BI_Raw								: FB_BA_BI_Raw := (
													iParent									:= B,
													sDescription							:= '{Sample BI (Raw Data)}',
													sDeviceType								:= 'Sicherung',
													sInactiveText							:= 'Normal',
													sActiveText								:= 'Ausgelöst',
													nEventClassID							:= MyECIDs.AlmStd
												);
		
			// Intention:						Input
			// Hardware:						I/O
			BI_DstbIO							: FB_BA_BI_IO := (
													iParent									:= B,
													sDescription							:= '{Sample BI Disturb (IO)}',
													sDeviceType								:= 'Sicherung',
													sInactiveText							:= 'Normal',
													sActiveText								:= 'Ausgelöst',
													ePolarity								:= E_BA_Polarity.eReverse,
													nEventClassID							:= MyECIDs.DstStd,
													eEnPlantLock							:= E_BA_LockPriority.eLocalMedium
												);
		
			// Intention:						Input for Display
			// Operation:						Display
			// Hardware:						I/O
			// Parameter:						EventDetectionEnable = FALSE
			BIDsp_SwiIO							: FB_BA_BI_IO := (
													iParent									:= B,
													sDescription							:= '{Sample BI Schalter Display (IO)}',
													sDeviceType								:= 'Sicherung',
													sInactiveText							:= 'Normal',
													sActiveText								:= 'Ausgelöst',
													ePolarity								:= E_BA_Polarity.eReverse,
													nEventClassID							:= MyECIDs.OthSmpl,
													bEventDetectionEnable					:= FALSE
												);
		
			// Intention:						Output
			// Hardware:						I/O
			BO_CmdIO							: FB_BA_BO_IO := (
													iParent									:= B,
													sDescription							:= '{Sample BO Befehl (IO)}',
													sInactiveText							:= 'Aus',
													sActiveText								:= 'Ein',
													nEventClassID							:= MyECIDs.AlmStd,
													stTimeDelay := (
														nToAbnormal							:= 3
													)
												);
		
			// Intention:						Output
			// Hardware:						Process Data
			BO_CmdProc							: FB_BA_BO := (
													iParent									:= B,
													sDescription							:= '{Sample BO Befehl (Process Data)}',
													sInactiveText							:= 'Aus',
													sActiveText								:= 'Ein',
													nEventClassID							:= MyECIDs.AlmStd,
													stTimeDelay := (
														nToAbnormal							:= 3
													)
												);
		
			// Intention:						Output
			// Hardware:						Raw Data
			BO_CmdRaw							: FB_BA_BO_Raw := (
													iParent									:= B,
													sDescription							:= '{Sample BO Befehl (Raw Data)}',
													sInactiveText							:= 'Aus',
													sActiveText								:= 'Ein',
													nEventClassID							:= MyECIDs.AlmStd,
													stTimeDelay := (
														nToAbnormal							:= 3
													)
												);
													
			// Intention:						Output for Display
			// Operation:						Display
			// Hardware:						I/O
			// Parameter:						EventDetectionEnable = FALSE
			BODisp_CmdIO						: FB_BA_BO_IO := (
													iParent									:= B,
													sDescription							:= '{Sample BO Befehl Display (IO)}',
													sInactiveText							:= 'Aus',
													sActiveText								:= 'Ein',
													nEventClassID							:= MyECIDs.OthSmpl,
													bEventDetectionEnable					:= FALSE
												);
	{endregion}
	{region 'Multistate'}
		M										: FB_BA_View := (
													iParent									:= THIS^,
													sDescription							:= '{Multistate objects}'
												);
			 
			// Intention:						Value
			MV									: FB_BA_MV := (
													iParent									:= M,
													sDescription							:= '{Sample MV}',
													aStateText								:= [ 'Aus', 'Stufe 1', 'Stufe 2' ],
													nEventClassID							:= MyECIDs.AlmStd
												);
			
			// Intention:						Value for Display
			// Operation:						Display
			nAVDsp_ValuePgm						: UDINT := 1;
			MVDsp								: FB_BA_MV_Op := (
													iParent									:= M,
													sObjectName								:= '{BAS01}',
													sDescription							:= '{Sample MV Display}',
													aStateText								:= [ 'Auto', 'Aus', 'Stufe 1', 'Stufe 2' ]
												);
			
			// Intention:						Value for Setpoint
			// Operation:						Setpoint
			MVSp								: FB_BA_MV_Op := (
													iParent									:= M,
													sObjectName								:= '{BAM01}',
													sDescription							:= '{Sample MV Setpoint}',
													aStateText								:= [ 'Auto', 'Aus', 'Stufe 1', 'Stufe 2' ],
													nValueRm								:= 1
												);
												
												
			nMVPushButton_Counter				: UDINT;
			MVPushButton						: FB_BA_MV_Op := (
													iParent									:= M,
													sDescription							:= '{Sample MV Pushbutton}',
													aStateText								:= [ 'Aus', 'Increment 1', 'Increment 2' ],
													eToggleMode								:= E_BA_ToggleMode.ePushButton
												);
		
			// Intention:						Input
			// Hardware:						Process Data
			MI_StateProc						: FB_BA_MI := (
													iParent									:= M,
													sDescription							:= '{Sample MI State (Process Data)}',
													sDeviceType								:= 'Gerät',
													aStateText								:= [ 'Aus', 'Stufe 1', 'Stufe 2', 'Stufe 3', 'Stufe 4' ],
													aAlarmValues							:= [ 3, 4 ],
													aFaultValues							:= [ 5 ],
													nEventClassID							:= MyECIDs.AlmStd
												);
		
			// Intention:						Input
			// Hardware:						Raw Data
			MI_StateRaw							: FB_BA_MI_Raw := (
													iParent									:= M,
													sDescription							:= '{Sample MI State (Raw Data)}',
													sDeviceType								:= 'Gerät',
													aStateText								:= [ 'Aus', 'Stufe 1', 'Stufe 2', 'Stufe 3', 'Stufe 4' ],
													aAlarmValues							:= [ 3, 4 ],
													aFaultValues							:= [ 5 ],
													nEventClassID							:= MyECIDs.AlmStd
												);
		
			// Intention:						Input
			// Hardware:						I/O
			MI_StateIO							: FB_BA_MI_IO := (
													iParent									:= M,
													sDescription							:= '{Sample MI State (IO)}',
													sDeviceType								:= 'Gerät',
													aStateText								:= [ 'Aus', 'Stufe 1', 'Stufe 2', 'Stufe 3', 'Stufe 4' ],
													aAlarmValues							:= [ 3, 4 ],
													aFaultValues							:= [ 5 ],
													nEventClassID							:= MyECIDs.AlmStd
												);
		
			// Intention:						Input for Display
			// Operation:						Display
			// Hardware:						I/O
			// Parameter:						EventDetectionEnable = FALSE
			MIDsp_Swi_StateIO					: FB_BA_MI_IO := (
													iParent									:= M,
													sDescription							:= '{Sample MI State (IO)}',
													sDeviceType								:= 'Gerät',
													aStateText								:= [ 'Zustand 1', 'Zustand 2', 'Zustand 3', 'Unbekannt' ],
													nEventClassID							:= MyECIDs.OthSmpl,
													bEventDetectionEnable					:= FALSE
												);
		
			// Intention:						Output for Display
			// Operation:						Display
			// Hardware:						I/O
			// Parameter:						EventDetectionEnable = FALSE
			MODisp_IO							: FB_BA_MO_IO := (
													iParent									:= M,
													sDescription							:= '{Sample MO Befehl (IO)}',
													aStateText								:= [ 'Aus', 'Stufe 1', 'Stufe 2', 'Stufe 3', 'Stufe 4' ],
													nEventClassID							:= MyECIDs.OthSmpl,
													bEventDetectionEnable					:= FALSE
												);
		
			// Intention:						Output
			// Hardware:						Process Data
			MO_CmdProc							: FB_BA_MO := (
													iParent									:= M,
													sDescription							:= '{Sample MO Befehl (Process Data)}',
													aStateText								:= [ 'Aus', 'Stufe 1', 'Stufe 2', 'Stufe 3', 'Stufe 4' ],
													nEventClassID							:= MyECIDs.OthSmpl
												);
		
			// Intention:						Output
			// Hardware:						Raw Data
			MO_CmdRaw							: FB_BA_MO_Raw := (
													iParent									:= M,
													sDescription							:= '{Sample MO Befehl (Raw Data)}',
													aStateText								:= [ 'Aus', 'Stufe 1', 'Stufe 2', 'Stufe 3', 'Stufe 4' ],
													nEventClassID							:= MyECIDs.OthSmpl
												);
	{endregion}
END_VAR

SUPER^();

// Analog:
A();

AV();
AVDsp(fValuePgm	:= MAX(fAVDsp_ValuePgm, AVSp.fPresentValue));
AVSp();
IF (bAVSp2_ValViaProp) THEN
	bAVSp2_ValViaProp := FALSE;
	AVSp2.PresentValue := fAVSp2_ValViaProp;
END_IF
AVSp2();
AI_Proc(fVal := fAI_Proc_ValuePgm);
AI_Raw();
AI_IO();
AI_IO_2_10V();
AI_Temp();
AIDsp_IO();
AO_CmdProc();
AO_CmdRaw();
AO_CmdIO();
AODisp_CmdIO();

// Binary:
B();

BV(bEnCrit := BI_DstbIO.bEvent);
BVDsp(bValuePgm	:= (bBVDsp_ValuePgm OR BVSp.bPresentValue));
BVSp();
BVPushButton();
BI_Proc();
BI_Raw();
BI_DstbIO();
BIDsp_SwiIO();
BO_CmdProc();
BO_CmdRaw();
BO_CmdIO();
BODisp_CmdIO();

IF (BVPushButton.bPresentValue <> BVPushButton.bDefaultValue) THEN
	nBVPushButton_Counter := (nBVPushButton_Counter+1);
END_IF

// Multistate:
M();

MV();
MVDsp(nValuePgm := MAX(nAVDsp_ValuePgm, MVSp.nPresentValue));
MVSp();
MVPushButton();
MI_StateProc();
MI_StateRaw();
MI_StateIO();
MIDsp_Swi_StateIO();
MODisp_IO(
	bEnPgm		:= TRUE,
	nValPgm		:= LIMIT(1, TO_UDINT(AVSp.fPresentValue), MODisp_IO.StateCount)
);
MO_CmdProc();
MO_CmdRaw();

IF (MVPushButton.nPresentValue <> MVPushButton.nDefaultValue) THEN
	nMVPushButton_Counter := (nMVPushButton_Counter+(MVPushButton.nPresentValue-1));
END_IF

END_FUNCTION_BLOCK

// ---- SAMPLES/Demo/Objects/FB_Obj_Misc.TcPOU
// Demonstration of objects.
// > See "FB_BA_EC01" to view decleared event classes.
FUNCTION_BLOCK FB_Obj_Misc EXTENDS FB_BA_View
VAR CONSTANT
	TREND_COUNT									: INT										:= 10;
END_VAR
VAR
	{region 'Project'}
		Proj									: FB_BA_View := (
													iParent									:= THIS^,
													sDescription							:= '{Project information}'
												);
				 
			// Intention:						Project Information
			Project								: FB_BA_Project := (
													iParent									:= Proj,
													sDescription							:= '{My project infos}',
													stProject := (	
														sTitle								:= 'Mein Projekt',
														sDescription						:= 'PLC Beispielprojekt',
														sLocation							:= 'Verl'
													)
												);
	{endregion}
	{region 'Loop'}
		Loop									: FB_BA_View := (
													iParent									:= THIS^,
													sDescription							:= '{Loop objects}'
												);
				 
			fLoop_Setpoint						: REAL										:= 20;								// Temperature setpoint.
			fLoop_CtrlVal						: REAL										:= 16;								// Simulation of controlled variable value.

			// Initialization:					Single loop for heating.
			Heat_En								: REFERENCE TO BOOL							REF= Heat.bEn;
			Heat_EnSync							: REFERENCE TO BOOL							REF= Heat.bEnSync;
			Heat_ValSync						: REFERENCE TO REAL							REF= Heat.fValSync;
			Heat_Y								: REFERENCE TO REAL							REF= Heat.fPresentValue;
			Heat								: FB_BA_LoopSeq := (
													iParent									:= Loop,
													sDescription							:= '{Heating Loop}',
													eOutputUnit								:= E_BA_Unit.eOther_Percent,
													bEn										:= TRUE,
													eActionRm								:= E_BA_Action.eReverse,
													fProportionalConstant					:= 3.0,
													fIntegralConstant						:= 180
												);

			// Initialization:					Single loop for heating.
			Cool_En								: REFERENCE TO BOOL							REF= Cool.bEn;
			Cool_EnSync							: REFERENCE TO BOOL							REF= Cool.bEnSync;
			Cool_ValSync						: REFERENCE TO REAL							REF= Cool.fValSync;
			Cool_Y								: REFERENCE TO REAL							REF= Cool.fPresentValue;
			Cool								: FB_BA_LoopSeq := (
													iParent									:= Loop,
													sDescription							:= '{Cooling Loop}',
													eOutputUnit								:= E_BA_Unit.eOther_Percent,
													bEn										:= TRUE,
													eActionRm								:= E_BA_Action.eDirect,
													fProportionalConstant					:= 3.0,
													fIntegralConstant						:= 180
												);
	{endregion}
	{region 'Calendar'}
		Cals									: FB_BA_View := (
													iParent									:= THIS^,
													sDescription							:= '{Calendar objects}'
												);

			// Intention:						Initialize calendar parameters with parameter builders.
			// Parameter:						tWeek										= F_BA_CalendarBuilder()
			Cal1								: FB_BA_Cal := (
													iParent									:= Cals,
													sDescription							:= '{Calendar 1}',
													aDateList								:= F_BA_CalendarBuilder()
																								.AppendDate(2021, E_BA_Month.eMarch, 10)
																								.AppendDateRange(nFromYear := 2021,E_BA_Month.eMarch,10, nToYear := 2021,E_BA_Month.eMarch,15)
																								.AppendWeekNDay(E_BA_Weekday.eMonday, E_BA_Week.Unspecified, E_BA_Month.Unspecified)
																								.Build()
												);
													 
			// Intention:						Initialize calendar parameters with helper methods.
			//									aDateList									= [(..., F_BA_DateVal(...)), (..., F_BA_DateRangeVal(...)), (..., F_BA_WeekNDayVal(...))]
			Cal2								: FB_BA_Cal := (
													iParent									:= Cals,
													sDescription							:= '{Calendar 2}',
													aDateList := [(
														eType								:= E_BA_DateValChoice.eDate,
														uDate								:= F_BA_DateVal(2020,E_BA_Month.eDecember,10)
													),(
														eType								:= E_BA_DateValChoice.eDateRange,
														uDate								:= F_BA_DateRangeVal(nFromYear:=2020,E_BA_Month.eMarch,5, nToYear:=2020,E_BA_Month.eMarch,10)
													),(
														eType								:= E_BA_DateValChoice.eWeekNDay,
														uDate								:= F_BA_WeekNDayVal(E_BA_Weekday.eTuesday, E_BA_Week.Unspecified, E_BA_Month.Unspecified)
													)]
												);

			Cal3								: FB_BA_Cal := (
													iParent									:= Cals,
													sDescription							:= '{Calendar 3}'
												);
	{endregion}
	{region 'Scheduler'}
		Sched									: FB_BA_View := (
													iParent									:= THIS^,
													sDescription							:= '{Schedule objects}'
												);
			
			// Intention:						Initialize scheduler parameters with parameter builders.
			// Parameter:						tWeek										= F_BA_WeeklyScheduleBuilder()
			//									tCalendar									= F_BA_ScheduleCalendarBuilder()
			//									tException									= F_BA_ExceptionScheduleBuilder()
			SchedA								: FB_BA_SchedA := (
													iParent									:= Sched,
													sDescription							:= '{Schedule Analog}',
													eUnit									:= E_BA_Unit.eTemperature_DegreesCelsius,
													aWeek									:= F_BA_WeeklyScheduleBuilder()
																								.SetAllDays()
																									.AppendA(T#0H, 1.0)
																									.Close()
																								.SetDay(E_BA_Weekday.eMonday)
																									.AppendA(T#0H, 2.0).AppendA(T#8H, 3.0).AppendA(T#16H, 2.0)
																									.Close()
																								.SetDayRange(E_BA_Weekday.eSaturday, E_BA_Weekday.eSunday)
																									.AppendA(T#0H, 4.0)
																									.Close()
																								.Build(),
													aCalendar								:= F_BA_ScheduleCalendarBuilder()
																								.AppendReference(Cal1)
																									.AppendA(T#0H, 1.0).AppendA(T#6H, 2.0).AppendNull(T#12H)
																									.Close()
																								.AppendReference(Cal2)
																									.AppendA(T#10H, 1.0).AppendNull(T#12H)
																									.Close()
																								.Build(),
													aException								:= F_BA_ExceptionScheduleBuilder()
																								.AppendDate(2021, E_BA_Month.eMarch, 10)
																									.AppendA(T#0H, 1.0).AppendA(T#6H, 2.0).AppendNull(T#12H)
																									.Close()
																								.AppendDateRange(nFromYear := 2021,E_BA_Month.eMarch,10, nToYear := 2021,E_BA_Month.eMarch,15)
																									.AppendA(T#12H, 1.0).AppendNull(T#16H)
																									.Close()
																								.AppendWeekNDay(E_BA_Weekday.eFriday, E_BA_Week.Unspecified, E_BA_Month.Unspecified)
																									.AppendA(T#20H, 3.0)
																									.Close()
																								.Build()
												);
			
			// Intention:						Initialize scheduler parameters with helper methods.
			// Parameter:						tWeek										= F_BA_SchedWeeklyXxA(...)
			//									tCalendar									= F_BA_SchedCalendar(...)
			//									tException									= [(..., F_BA_SchedEntryXxA(...)), (..., F_BA_SchedEntryXxA(...)), (..., F_BA_SchedEntryXxA(...))]
			SchedB								: FB_BA_SchedB := (
													iParent									:= Sched,
													sDescription							:= '{Schedule Bool}',
													sInactiveText							:= 'Aus',
													sActiveText								:= 'Ein',
													aWeek									:= F_BA_SchedWeekly3xB(E_BA_Weekday.eMonday, E_BA_Weekday.eFriday, T#0H, FALSE, T#6H, TRUE, T#20H, FALSE),
													aCalendar := [(
														iRefCalendar						:= Cal1,
														aEntry								:= F_BA_SchedEntry2xB(T#8H, TRUE, T#18H, FALSE)
													)],
													aException := [(
														eType								:= E_BA_DateValChoice.eDate,
														uDate								:= F_BA_DateVal(2021,E_BA_Month.eMarch,10),
														aEntry								:= F_BA_SchedEntry1xB(T#0H, FALSE)
													),(
														eType								:= E_BA_DateValChoice.eDateRange,
														uDate								:= F_BA_DateRangeVal(nFromYear:=2021,E_BA_Month.eMarch,10, nToYear:=2021,E_BA_Month.eMarch,15),
														aEntry								:= F_BA_SchedEntry2xB(T#10H, TRUE, T#17H, F_BA_NullB())
													),(
														eType								:= E_BA_DateValChoice.eWeekNDay,
														uDate								:= F_BA_WeekNDayVal(E_BA_Weekday.eFriday, E_BA_Week.Unspecified, E_BA_Month.Unspecified),
														aEntry								:= F_BA_SchedEntry3xB(T#9H, FALSE, T#12H, TRUE, T#17H, F_BA_NullB())
													)]);
			// Intention:						Initialize scheduler parameters manually.
			//									tCalendar									= ...
			//									tException									= ...
			SchedM								: FB_BA_SchedM := (
													iParent									:= Sched,
													sDescription							:= '{Schedule Multistate}',
													aStateText								:= [ 'Aus', 'Stufe 1', 'Stufe 2', 'Stufe 3' ],
													aWeek									:= F_BA_SchedWeekly3xM(E_BA_Weekday.eMonday, E_BA_Weekday.eFriday, T#0H, 1, T#6H, 2, T#20H, 1),
													aCalendar := [(
														iRefCalendar						:= Cal1,
														aEntry := [(
															eState							:= E_BA_SchedEntryState.eValue,
															stTime							:= F_BA_ToSTTime(T#16H),
															uValue							:= F_BA_UDIVal(2)
														),(
															eState							:= E_BA_SchedEntryState.eValue,
															stTime							:= F_BA_ToSTTime(T#20H),
															uValue							:= F_BA_UDIVal(1)
														)]
													)],
													aException := [(
														eType								:= E_BA_DateValChoice.eWeekNDay,
														uDate								:= F_BA_WeekNDayVal(E_BA_Weekday.eFriday, E_BA_Week.Unspecified, E_BA_Month.Unspecified),
														aEntry := [(
															eState							:= E_BA_SchedEntryState.eValue,
															stTime							:= F_BA_ToSTTime(T#10H),
															uValue							:= F_BA_UDIVal(2)
														),(
															eState							:= E_BA_SchedEntryState.eValue,
															stTime							:= F_BA_ToSTTime(T#12H),
															uValue							:= F_BA_UDIVal(3)
														),(
															eState							:= E_BA_SchedEntryState.eNull,
															stTime							:= F_BA_ToSTTime(T#16H)
														)]
													)]);
	{endregion}
	{region 'Trend'}
		Trnd									: FB_BA_View := (
													iParent									:= THIS^,
													sDescription							:= '{Trend objects}'
												);
				 
			// Intention:						Trend in polling-mode
			// Parameter:						eLoggingType								= E_BA_LoggingType.ePolled
			PollAV								: FB_BA_AV_Op := (
													iParent									:= Trnd,
													sDescription							:= '{Referenced object for polling}',
													eUnit									:= E_BA_Unit.eTemperature_DegreesCelsius,
													fValueRm								:= 3
												);
			TrendPoll							: FB_BA_Trend := (
													iParent									:= Trnd,
													sDescription							:= '{Sample Trend}',
													nEventClassID							:= MyECIDs.AlmStd,
													bEnable									:= TRUE,
													stStartTime								:= F_BA_ToSTDateTime(DT#2010-01-01-00:00),
													eLoggingType							:= E_BA_LoggingType.ePolled,
													nLogInterval							:= 300,
													stReferencedParam							:= F_BA_Reference(PollAV, E_BA_Parameter.ePresentValue)
												);
													
			// Intention:						Trend in trigger-mode
			// Parameter:						eLoggingType								= E_BA_LoggingType.ePolled
			TrigAV								: FB_BA_AV_Op := (
													iParent									:= Trnd,
													sDescription							:= '{Referenced object for polling}',
													eUnit									:= E_BA_Unit.eTemperature_DegreesCelsius,
													fValueRm								:= 1
												);
			TrendTrig_Man						: BOOL;
			TrendTrig							: FB_BA_Trend := (
													iParent									:= Trnd,
													sDescription							:= '{Sample Trend}',
													nEventClassID							:= MyECIDs.AlmStd,
													bEnable									:= TRUE,
													stStartTime								:= F_BA_ToSTDateTime(DT#2010-01-01-00:00),
													eLoggingType							:= E_BA_LoggingType.eTriggered,
													stReferencedParam						:= F_BA_Reference(TrigAV, E_BA_Parameter.ePresentValue)
												);
													 
			// Intention:						Trend in COV-mode
			// Parameter:						eLoggingType								= E_BA_LoggingType.eCOV
			CovAI								: FB_BA_AI := (
													iParent									:= Trnd,
													sDescription							:= '{Referenced analog object for COV}',
													eUnit									:= E_BA_Unit.eOther_Percent,
													nEventClassID							:= MyECIDs.AlmStd,
													bEventDetectionEnable					:= FALSE
												);
			TrendCovAI							: FB_BA_Trend := (
													iParent									:= Trnd,
													sDescription							:= '{Sample Analog Trend COV}',
													nEventClassID							:= MyECIDs.AlmStd,
													bEnable									:= TRUE,
													nBufferSize								:= 100,
													eLoggingType							:= E_BA_LoggingType.eCOV,
													stReferencedParam							:= F_BA_Reference(CovAI, E_BA_Parameter.ePresentValue)
												);
			CovBI								: FB_BA_BI := (
													iParent									:= Trnd,
													sDescription							:= '{Referenced binary object for COV}',
													sInactiveText							:= 'Off',
													sActiveText								:= 'On',
													nEventClassID							:= MyECIDs.AlmStd,
													bEventDetectionEnable					:= FALSE
												);
			TrendCovBI							: FB_BA_Trend := (
													iParent									:= Trnd,
													sDescription							:= '{Sample Binary Trend COV}',
													nEventClassID							:= MyECIDs.AlmStd,
													bEnable									:= TRUE,
													nBufferSize								:= 100,
													eLoggingType							:= E_BA_LoggingType.eCOV,
													stReferencedParam						:= F_BA_Reference(CovBI, E_BA_Parameter.ePresentValue)
												);
			CovMI								: FB_BA_MI := (
													iParent									:= Trnd,
													sDescription							:= '{Referenced multistate object for COV}',
													aStateText								:= ['Eco', 'Standard', 'Comfort'],
													nEventClassID							:= MyECIDs.AlmStd,
													bEventDetectionEnable					:= FALSE
												);
			TrendCovMI							: FB_BA_Trend := (
													iParent									:= Trnd,
													sDescription							:= '{Sample Multistate Trend COV}',
													nEventClassID							:= MyECIDs.AlmStd,
													bEnable									:= TRUE,
													nBufferSize								:= 100,
													eLoggingType							:= E_BA_LoggingType.eCOV,
													stReferencedParam						:= F_BA_Reference(CovMI, E_BA_Parameter.ePresentValue)
												);
													 
			// Intention:						Multiple trend objects as array
			Trends								: FB_BA_View := (
													iParent									:= Trnd,
													sDescription							:= 'Multiple trend objects'
												);
				Trend							: ARRAY[1 .. TREND_COUNT] OF FB_BA_Trend := [TREND_COUNT((
													iParent									:= Trends,
													iLabel									:= MyLabels.Trnd,
													nEventClassID							:= MyECIDs.AlmStd,
													eLoggingType							:= E_BA_LoggingType.eCOV
												))];
	{endregion}
END_VAR
VAR			
	_i											: INT;
END_VAR

SUPER^();

// Project:
Proj();

Project();

// Calendar:
Cals();

Cal1();
Cal2();
Cal3();

// Scheduler:
Sched();

SchedA();
SchedB();
SchedM();

// Loop:
Loop();

Heat(
	fSetpoint := fLoop_Setpoint,
	fCtrlVal := fLoop_CtrlVal
);
Cool(
	fSetpoint := fLoop_Setpoint,
	fCtrlVal := fLoop_CtrlVal
);

// Trend:
Trnd();

PollAV();
TrendPoll();
TrigAV(fValuePgm:=(TrigAV.fValuePgm+0.01));
TrendTrig(bTrigPgm:=((MAIN.nCounter MOD 250 = 0) OR (TrendTrig_Man)));
IF (MAIN.nCounter MOD 200 = 0) THEN
	CovAI.fVal := SEL((CovAI.fVal<10), 0, (CovAI.fVal+1));
END_IF
IF (MAIN.nCounter MOD 500 = 0) THEN
	CovBI.bVal := (NOT CovBI.bVal);
	CovMI.nVal := SEL((CovMI.nVal<CovMI.StateCount), 1, (CovMI.nVal+1));
END_IF
CovAI();
TrendCovAI();
CovBI();
TrendCovBI();
CovMI();
TrendCovMI();
Trends();
FOR _i := 1 TO TREND_COUNT DO
	Trend[_i]();
END_FOR

END_FUNCTION_BLOCK

// ---- SAMPLES/MAIN.TcPOU
PROGRAM MAIN
VAR
	{region 'Settings'}
		DPAD						: FB_BA_CarelessDPAD:=(
										aIdentifier:=[
											(* Level 1 *)	(eNodeType:=E_BA_NodeType.eBuilding,	nIndexDigits:=2),
											(* Level 2 *)	(eNodeType:=E_BA_NodeType.eTrade,		nIndexDigits:=0),
											(* Level 3 *)	(eNodeType:=E_BA_NodeType.ePlant,		nIndexDigits:=2,			sSeparator_ObjectName:='~~~',		sSeparator_Description:=' --- '),
											(* Level 4 *)	(eNodeType:=E_BA_NodeType.eAggregate,	nIndexDigits:=2,			sSeparator_ObjectName:='++'),
											(* Level 5 *)	(eNodeType:=E_BA_NodeType.eFunction,	nIndexDigits:=3)
									]);
	{endregion}
		 
	Smpl							: FB_BA_View			:= (									sDescription:='Samples');
	{region 'Demonstration'}
		Demo						: FB_BA_View			:= (iParent:=Smpl,						sDescription:='Demonstration');
			Obj						: FB_BA_View			:= (iParent:=Demo,						sDescription:='Objects');
				General				: FB_Obj_General		:= (iParent:=Obj,						sDescription:='General objects');
				Misc				: FB_Obj_Misc			:= (iParent:=Obj,						sDescription:='Miscellaneous objects');
				Seq					: FB_Obj_Sequence		:= (iParent:=Obj,						sDescription:='Sequences');
				UdObj				: FB_Obj_UserDefined	:= (iParent:=Obj,						sDescription:='User defined objects');
				AddParam			: FB_Obj_AddParam		:= (iParent:=Obj,						sDescription:='Additional parameters');

			Ref						: FB_BA_View			:= (iParent:=Demo,						sDescription:='Reference');
				Collect				: FB_Ref_Collectors		:= (iParent:=Ref,						sDescription:='Collectors');
				Groups				: FB_Ref_Groups			:= (iParent:=Ref,						sDescription:='Groups');
				PubSubLc			: FB_Ref_PubSub_Local	:= (iParent:=Ref,						sDescription:='Publisher and subscriber (Local)');
				PubSubRm			: FB_Ref_PubSub_Remote	:= (iParent:=Ref,						sDescription:='Publisher and subscriber (Remote)');

			Evt						: FB_BA_View			:= (iParent:=Demo,						sDescription:='Event');
				EvtCls				: FB_Evt_EventClasses	:= (iParent:=Evt,						sDescription:='Event classes');
				Events				: FB_Evt_Events			:= (iParent:=Evt,						sDescription:='Events');
				Ack					: FB_Evt_Ack			:= (iParent:=Evt,						sDescription:='Acknowledgement');
				MiscEvt				: FB_Evt_Misc			:= (iParent:=Evt,						sDescription:='Miscellaneous');
				Cnd					: FB_Evt_QueryCnd;

			Strct					: FB_BA_View			:= (iParent:=Demo,						sDescription:='Structure');
				Nested				: FB_Struct_Nested		:= (iParent:=Strct,						sDescription:='Nested objects');

			Plt						: FB_BA_View			:= (iParent:=Demo,						sDescription:='Plant');
				PltCtrl1			: FB_Plt_Init1			:= (iParent:=Plt,						sDescription:='Plant control initialization 1');
				PltCtrl2			: FB_Plt_Init2			:= (iParent:=Plt,						sDescription:='Plant control initialization 2');
				PltCtrl3			: FB_Plt_Init3			:= (iParent:=Plt,						sDescription:='Plant control initialization 3');

			Spl						: FB_BA_View			:= (iParent:=Demo,						sDescription:='Supplement specific');
				BACnet_RcpList		: FB_BACnet_RcpList		:= (iParent:=Spl,						sDescription:='Write Recipient list (BACnet)');
				BACnet_ObjPropRef	: FB_BACnet_ObjPropRef	:= (iParent:=Spl,						sDescription:='Write object property reference (BACnet)');
				BACnet_EvtInh		: FB_BACnet_EvtInh		:= (iParent:=Spl,						sDescription:='Write EventInhibit property (BACnet)');
					 
			Other					: FB_BA_View			:= (iParent:=Demo,						sDescription:='Other');
				Texts				: FB_Texts				:= (iParent:=Other,						sDescription:='Name and description texts');
				MscOth				: FB_Misc				:= (iParent:=Other,						sDescription:='Miscellaneous');
	{endregion}
	{region 'Templates'}
		Tmpl						: FB_BA_View			:= (iParent:=Smpl,						sDescription:='Templates');
			Gen						: FB_BA_View			:= (iParent:=Tmpl,						sDescription:='General');
				Bld01				: FB_BA_Bld01			:= (iParent:=Gen,						sDescription:='Building information');
				EvtCls01			: FB_BA_EC01			:= (iParent:=Gen,						sDescription:='Event Classes');
	{endregion}		
END_VAR
VAR		
	nCounter						: UDINT					:= 0;	
END_VAR

nCounter:=(nCounter+1);

Smpl();

// Demonstration:
Demo();

Obj();
General();
Misc();
Seq();
UdObj();
AddParam();

Ref();
Collect();
Groups();
PubSubLc();
PubSubRm();

Evt();
EvtCls();
Events();
Ack();
MiscEvt();
Cnd();

Strct();
Nested();

Plt();
PltCtrl1();
PltCtrl2();
PltCtrl3();

Spl();
BACnet_RcpList();
BACnet_ObjPropRef();
BACnet_EvtInh();

Other();
Texts();
MscOth();

// Templates:
Tmpl();

Gen();
Bld01();
EvtCls01();

// Optional extensions:
MAIN_OPTEXT();
MAIN_OPTEXT_BACnet();

END_PROGRAM

// ---- SAMPLES/Demo/Reference/Publish and Subscribe/FB_Ref_PubSub_Remote.TcPOU
// Example of "device-to-device" communication.
// [Notes]
// > Apply devices routes via "Diangnose / Device communication" in Site Explorer when PLC's are in run-mode.
//   Afterwards all communication errors will disappear. 
FUNCTION_BLOCK FB_Ref_PubSub_Remote EXTENDS FB_BA_View
VAR CONSTANT
	{region 'Test Settings'}
		// Use one (remote) device:
//		sDevice1_NetID			: T_BA_MedString				:= '192.168.10.100.1.1';
//		sDevice2_NetID			: T_BA_MedString				:= '192.168.10.100.1.1';
			 
		// Use one (loopback) device:
		sDevice1_NetID			: T_BA_MedString				:= '127.0.0.1.1.1';
		sDevice2_NetID			: T_BA_MedString				:= '127.0.0.1.1.1';
			 
		// Use two (remote and loopback) devices:
//		sDevice1_NetID			: T_BA_MedString				:= '192.168.2.200.1.1';
//		sDevice2_NetID			: T_BA_MedString				:= '127.0.0.1.1.1';
			 
		// Use two (remote) devices:
//		sDevice1_NetID			: T_BA_MedString				:= '192.168.10.100.1.1';
//		sDevice2_NetID			: T_BA_MedString				:= '192.168.2.200.1.1';
	{endregion}
END_VAR
VAR
	{region 'Analog'}
		AV_Sub					: FB_BA_SubAPrio := (
									sSubject					:= 'AV_Obj',
									sTarget						:= sDevice1_NetID,
									tReadInterval				:= T#5S								// Set shorter read interval
								);
		AVOp_Sub				: FB_BA_SubAV_Op := (
									sSubject					:= 'AVOp_Obj',
									sTarget						:= sDevice1_NetID,
									tReadInterval				:= T#5S								// Set shorter read interval
								);
		AI_Sub					: FB_BA_SubAI := (
									sSubject					:= 'AI_Obj',
									sTarget						:= sDevice2_NetID,
									tReadInterval				:= T#5S								// Set shorter read interval
								);
		AO_Sub					: FB_BA_SubAPrio := (
									sSubject					:= 'AO_Obj',
									sTarget						:= sDevice2_NetID,
									tReadInterval				:= T#5S								// Set shorter read interval
								);
	{endregion}
	{region 'Binary'}
		BV_Sub					: FB_BA_SubBPrio := (
									sSubject					:= 'BV_Obj',
									sTarget						:= sDevice1_NetID
								);
		BVOp_Sub				: FB_BA_SubBV_Op := (
									sSubject					:= 'BVOp_Obj',
									sTarget						:= sDevice1_NetID
								);
		BI_Sub					: FB_BA_SubBI := (
									sSubject					:= 'BI_Obj',
									sTarget						:= sDevice2_NetID
								);
		BO_Sub					: FB_BA_SubBPrio := (
									sSubject					:= 'BO_Obj',
									sTarget						:= sDevice2_NetID
								);
	{endregion}
	{region 'Multistate'}
		MV_Sub					: FB_BA_SubMPrio := (
									sSubject					:= 'MV_Obj',
									sTarget						:= sDevice1_NetID
								);
		MVOp_Sub				: FB_BA_SubMV_Op := (
									sSubject					:= 'MVOp_Obj',
									sTarget						:= sDevice1_NetID
								);
		MI_Sub					: FB_BA_SubMI := (
									sSubject					:= 'MI_Obj',
									sTarget						:= sDevice2_NetID
								);
		MO_Sub					: FB_BA_SubMPrio := (
									sSubject					:= 'MO_Obj',
									sTarget						:= sDevice2_NetID
								);
	{endregion}
	{region 'Multistate'}
		Loop_Sub				: FB_BA_SubLoop := (
									sSubject					:= 'Loop_Obj',
									sTarget						:= sDevice1_NetID
								);		
		Cal_Sub					: FB_BA_SubCal := (
									sSubject					:= 'Cal_Obj',
									sTarget						:= sDevice1_NetID
								);
		SchedA_Sub				: FB_BA_SubSchedA := (
									sSubject					:= 'SchedA_Obj',
									sTarget						:= sDevice1_NetID
								);
		SchedB_Sub				: FB_BA_SubSchedB := (
									sSubject					:= 'SchedB_Obj',
									sTarget						:= sDevice1_NetID
								);
		SchedM_Sub				: FB_BA_SubSchedM := (
									sSubject					:= 'SchedM_Obj',
									sTarget						:= sDevice1_NetID
								);
		Trend_Sub				: FB_BA_SubTrend := (
									sSubject					:= 'Trend_Obj',
									sTarget						:= sDevice2_NetID
								);
	{endregion}	  
	{region 'Custom'}
		{region 'Typed'}  
			MyWthSt1_Sub		: FB_BA_MyWeatherStationSub := (
									sSubject					:= 'MyWthSt',
									sTarget						:= sDevice1_NetID,
									tReadInterval				:= T#5S,							// Set shorter read interval
									tReadTolerance				:= T#20S,							// Tolerate read errors for a short time
									bClearOnReadError			:= TRUE								// Clear data on error
								);
			MyWthSt2_Sub		: FB_BA_MyWeatherStationSub := (
									sSubject					:= 'MyWthSt',
									sTarget						:= sDevice2_NetID
								);
			MyWthSt3_Sub		: FB_BA_MyWeatherStationSub := (
									sSubject					:= 'MyWthSt',
									sTarget						:= sDevice2_NetID
								);
		{endregion}
		{region 'Raw'}
			MyRawWthSt1Data_Sub	: ST_BA_MyWeatherData;
			MyRawWthSt1_Sub		: FB_BA_RawSubscriber := (
									sSubject					:= 'MyRawWthSt',
									sTarget						:= sDevice1_NetID
								);
			MyRawWthSt2Data_Sub	: ST_BA_MyWeatherData;
			MyRawWthSt2_Sub		: FB_BA_RawSubscriber := (
									sSubject					:= 'MyRawWthSt',
									sTarget						:= sDevice2_NetID
								);
		{endregion}
	{endregion} 
	{region 'Tests'}
		{region 'Subject path'}
			Nested1a_AV_Sub		: FB_BA_SubAV_Op := (
								//	sSubject					:= 'fbAV',							// -> Would lead to ambiguous subject!
									sSubject					:= 'Nested1a.Value',
									sTarget						:= sDevice1_NetID
								);
			Nested1b_AV_Sub		: FB_BA_SubAV_Op := (
								//	sSubject					:= 'fbAV',							// -> Would lead to ambiguous subject!
									sSubject					:= 'Nested1b.Value',
									sTarget						:= sDevice1_NetID
								);
		{endregion}
	{endregion}
END_VAR

SUPER^(); // FB_BA_View
AO_Sub(); // FB_BA_SubAPrio
AV_Sub(); // FB_BA_SubAPrio
AVOp_Sub(); // FB_BA_SubAV_Op
AI_Sub(); // FB_BA_SubAI
MyWthSt3_Sub(); // FB_BA_MyWeatherStationSub
BO_Sub(); // FB_BA_SubBPrio
BV_Sub(); // FB_BA_SubBPrio
BVOp_Sub(); // FB_BA_SubBV_Op
BI_Sub(); // FB_BA_SubBI
MO_Sub(); // FB_BA_SubMPrio
MV_Sub(); // FB_BA_SubMPrio
MVOp_Sub(); // FB_BA_SubMV_Op
MI_Sub(); // FB_BA_SubMI
Loop_Sub(); // FB_BA_SubLoop
Cal_Sub(); // FB_BA_SubCal
SchedA_Sub(); // FB_BA_SubSchedA
SchedB_Sub(); // FB_BA_SubSchedB
SchedM_Sub(); // FB_BA_SubSchedM
Trend_Sub(); // FB_BA_SubTrend
Nested1a_AV_Sub(); // FB_BA_SubAV_Op
MyRawWthSt1_Sub(xData := MyRawWthSt1Data_Sub); // FB_BA_RawSubscriber
MyWthSt1_Sub(); // FB_BA_MyWeatherStationSub
Nested1b_AV_Sub(); // FB_BA_SubAV_Op
MyWthSt2_Sub(); // FB_BA_MyWeatherStationSub
MyRawWthSt2_Sub(xData := MyRawWthSt2Data_Sub); // FB_BA_RawSubscriber

END_FUNCTION_BLOCK

// ---- SAMPLES/Demo/Supplement specific/BACnet/FB_BACnet_RcpList.TcPOU
// Exemple illustrates how to write the (BACnet) recipient list to a 'FB_BA_EC' object.
FUNCTION_BLOCK FB_BACnet_RcpList EXTENDS FB_BA_View
VAR
	bWrite				: BOOL;
	
	// Recipient list to write (to all event classes):
	aRecipientList		: T_BACnet_RecipientList := [(
							nProcessId					:= 20100,
							stValidDays					:= F_BACnet_ValidDays(TRUE, TRUE, TRUE, TRUE, TRUE, TRUE, TRUE),
							stFromTime					:= F_BA_ToSTTime(T#0H),
							stToTime					:= F_BA_ToSTTime(T#23H59M59S),
							bIssueConfirmed				:= FALSE,
							stEventTransitions			:= F_BACnet_EventTransitionBits(TRUE, TRUE, TRUE),
							stRecipient					:= F_BACnet_DeviceRecipient(nDeviceInstance:=5)
						),(
							nProcessId					:= 30100,
							stValidDays					:= F_BACnet_ValidDays(TRUE, TRUE, TRUE, TRUE, TRUE, FALSE, FALSE),
							stFromTime					:= F_BA_ToSTTime(T#0H),
							stToTime					:= F_BA_ToSTTime(T#23H59M59S),
							bIssueConfirmed				:= TRUE,
							stEventTransitions			:= F_BACnet_EventTransitionBits(TRUE, TRUE, TRUE),
							stRecipient					:= F_BACnet_EthernetRecipient(nIPAddress1:=192,168,10,200, nPort:=47808, nNetworkNr:=444)
						)];
END_VAR
VAR
	_iObj				: I_BA_Object;
	_fbBACnetObj		: POINTER TO FB_BACnet_BaseObject;
	_hRes				: HRESULT;
END_VAR

SUPER^();

IF (bWrite) THEN
	bWrite := FALSE;
	
	// Iterate over all event class objects:
	_iObj := 0;
	WHILE (F_BA_IterateObjectIndex(_iObj, E_BA_ObjectType.eEventClass)) DO
		// Receive internal BACnet object from BA object:
		IF (NOT _iObj.GetBACnetObject(fbObject=>_fbBACnetObj)) THEN
			_iObj.LogMsg.Show(ADSLOG_MSGTYPE_ERROR, 'RL09', 'Failed to receive internal BACnet object!', TRUE);
		ELSE
			// Write recipient list:
			_hRes := _fbBACnetObj^.WritePropertyRecipientList(aRecipientList);
			IF (FAILED(_hRes)) THEN
				; // Do some error handling (An error message has already been logged here).
			END_IF
		END_IF
	END_WHILE
END_IF

END_FUNCTION_BLOCK

// ---- SAMPLES/Demo/Supplement specific/BACnet/FB_BACnet_EvtInh.TcPOU
// Exemple illustrates how to write the 'EventAlgotithmInhibit' BACnet property of event enabled objects.
FUNCTION_BLOCK FB_BACnet_EvtInh EXTENDS FB_BA_View
VAR
	bWrite			: BOOL;
	bValue			: BOOL				:= TRUE;
END_VAR
VAR
	_iObj			: I_BA_Object;
	_fbBACnetObj	: POINTER TO FB_BACnet_BaseObject;
	_hRes			: HRESULT;
END_VAR

SUPER^();

IF (bWrite) THEN
	bWrite := FALSE;
	
	// Iterate over all objects:
	_iObj := 0;
	WHILE (F_BA_IterateObjects(_iObj)) DO	
		// Iterate over all EventObjects:	     
		IF (_iObj.EventAbility <> E_BA_EventAbility.eEventEx) THEN
			; // Skip.
		ELSIF (NOT _iObj.GetBACnetObject(fbObject=>_fbBACnetObj)) THEN
			_iObj.LogMsg.Show(ADSLOG_MSGTYPE_ERROR, 'EI13', 'Failed to receive internal BACnet object!', TRUE);
		ELSE
			// Enable and write property:
			_hRes := _fbBACnetObj^.WritePropertyBool(E_BACnetPropIdentifier.PropEventAlgorithmInhibit, bValue);
			IF (FAILED(_hRes)) THEN
				; // Do some error handling (An error message has already been logged here).
			END_IF
		END_IF
	END_WHILE
	
	// [Alternative]
	// Iterate over all child-objects of this current view: 
	(*
	WHILE (THIS^.IterateObjects(_iObj)) DO
		// ...
	END_WHILE
	*)
END_IF

END_FUNCTION_BLOCK

// ---- SAMPLES/Templates/Standard/POUs/Trade/General/Building/FB_BA_Bld01.TcPOU
FUNCTION_BLOCK FB_BA_Bld01 EXTENDS FB_BA_View
VAR
	FireAlarm		: FB_BA_BV_OP := (
						iParent					:= THIS^,
						sDescription			:= 'Fire Alarm',
						sInactiveText			:= 'Inaktiv',
						sActiveText				:= 'Aktiv',
						bValueRm				:= FALSE);
						
	BurglarAlarm	: FB_BA_BV_OP := (
						iParent					:= THIS^,
						sDescription			:= 'Burglar Alarm',
						sInactiveText			:= 'Inaktiv',
						sActiveText				:= 'Aktiv',
						bValueRm				:= FALSE);
						
	IceAlarm		: FB_BA_BV_OP := (
						iParent					:= THIS^,
						sDescription			:= 'Ice Alarm',
						sInactiveText			:= 'Inaktiv',
						sActiveText				:= 'Aktiv',
						bValueRm				:= FALSE);
						
	Maintenance		: FB_BA_BV_OP := (
						iParent					:= THIS^,
						sDescription			:= 'Maintenance',
						sInactiveText			:= 'Inaktiv',
						sActiveText				:= 'Aktiv',
						bValueRm				:= FALSE);
						
	StormProtection	: FB_BA_BV_OP := (
						iParent					:= THIS^,
						sDescription			:= 'Storm Protection',
						sInactiveText			:= 'Inaktiv',
						sActiveText				:= 'Aktiv',
						bValueRm				:= FALSE);
						
	SunProtection	: FB_BA_BV_OP := (
						iParent					:= THIS^,
						sDescription			:= 'Sun Protection',
						sInactiveText			:= 'Inaktiv',
						sActiveText				:= 'Aktiv',
						bValueRm				:= FALSE);
						
	ThermalAutomatic: FB_BA_BV_OP := (
						iParent					:= THIS^,
						sDescription			:= 'Thermal Automatic',
						sInactiveText			:= 'Inaktiv',
						sActiveText				:= 'Aktiv',
						bValueRm				:= FALSE);
END_VAR

SUPER^();

FireAlarm();
BurglarAlarm();
IceAlarm();
Maintenance();
StormProtection();
SunProtection();
ThermalAutomatic();

END_FUNCTION_BLOCK

// ---- SAMPLES/Templates/Standard/POUs/Trade/General/EventClasses/FB_BA_EC01.TcPOU
// Template of event classes.
FUNCTION_BLOCK FB_BA_EC01 EXTENDS FB_BA_View
VAR CONSTANT
	OBJECT_NAME			: STRING					:= 'EC{InstID}';
END_VAR
VAR
	{region 'Alarm'}
		AlmSmpl			: FB_BA_EC := (
							iParent					:= THIS^,
							nInstanceID				:= 12,
							sObjectName				:= OBJECT_NAME,
							sDescription			:= '{Alarm (Einfach)}',
							eEventType				:= E_BA_EventType.eAlarm,
							eAlarmMode				:= E_BA_AlarmMode.eSimple,
							aPriority				:= [ 10, 11, 12 ]
						);
		AlmStd			: FB_BA_EC := (
							iParent					:= THIS^,
							nInstanceID				:= 11,
							sObjectName				:= OBJECT_NAME,
							sDescription			:= '{Alarm (Standard)}',
							eEventType				:= E_BA_EventType.eAlarm,
							eAlarmMode				:= E_BA_AlarmMode.eStandard,
							aPriority				:= [ 13, 14, 15 ]
						);
		AlmExt			: FB_BA_EC := (
							iParent					:= THIS^,
							nInstanceID				:= 10,
							sObjectName				:= OBJECT_NAME,
							sDescription			:= '{Alarm (Erweitert)}',
							eEventType				:= E_BA_EventType.eAlarm,
							eAlarmMode				:= E_BA_AlarmMode.eExtended,
							aPriority				:= [ 16, 17, 18 ]
						);
	{endregion}
	{region 'Disturb'}
		DstSmpl			: FB_BA_EC	:= (
							iParent					:= THIS^,
							nInstanceID				:= 52,
							sObjectName				:= OBJECT_NAME,
							sDescription			:= '{Störung (Einfach)}',
							eEventType				:= E_BA_EventType.eDisturb,
							eAlarmMode				:= E_BA_AlarmMode.eSimple,
							aPriority				:= [ 50, 51, 52 ]
						);
		DstStd			: FB_BA_EC := (
							iParent					:= THIS^,
							nInstanceID				:= 51,
							sObjectName				:= OBJECT_NAME,
							sDescription			:= '{Störung (Standard)}',
							eEventType				:= E_BA_EventType.eDisturb,
							eAlarmMode				:= E_BA_AlarmMode.eStandard,
							aPriority				:= [ 53, 54, 55 ]
						);
		DstExt			: FB_BA_EC := (
							iParent					:= THIS^,
							nInstanceID				:= 50,
							sObjectName				:= OBJECT_NAME,
							sDescription			:= '{Störung (Erweitert)}',
							eEventType				:= E_BA_EventType.eDisturb,
							eAlarmMode				:= E_BA_AlarmMode.eExtended,
							aPriority				:= [ 56, 57, 58 ]
						);
	{endregion}
	{region 'Maintenance'}
		MntnSmpl		: FB_BA_EC := (
							iParent					:= THIS^,
							nInstanceID				:= 92,
							sObjectName				:= OBJECT_NAME,
							sDescription			:= '{Wartung (Einfach)}',
							eEventType				:= E_BA_EventType.eMaintenance,
							eAlarmMode				:= E_BA_AlarmMode.eSimple,
							aPriority				:= [ 90, 91, 92 ]
						);
		MntnStd			: FB_BA_EC := (
							iParent					:= THIS^,
							nInstanceID				:= 91,
							sObjectName				:= OBJECT_NAME,
							sDescription			:= '{Wartung (Standard)}',
							eEventType				:= E_BA_EventType.eMaintenance,
							eAlarmMode				:= E_BA_AlarmMode.eStandard,
							aPriority				:= [ 93, 94, 95 ]
						);

		MntnExt			: FB_BA_EC := (
							iParent					:= THIS^,
							nInstanceID				:= 90,
							sObjectName				:= OBJECT_NAME,
							sDescription			:= '{Wartung (Erweitert)}',
							eEventType				:= E_BA_EventType.eMaintenance,
							eAlarmMode				:= E_BA_AlarmMode.eExtended,
							aPriority				:= [ 96, 97, 98 ]
						);
	{endregion}
	{region 'Notification'}
		NtfSmpl			: FB_BA_EC := (
							iParent					:= THIS^,
							nInstanceID				:= 132,
							sObjectName				:= OBJECT_NAME,
							sDescription			:= '{Benachrichtigung (Einfach)}',
							eEventType				:= E_BA_EventType.eNotification,
							eAlarmMode				:= E_BA_AlarmMode.eSimple,
							aPriority				:= [ 130, 131, 132 ]
						);
		NtfStd			: FB_BA_EC := (
							iParent					:= THIS^,
							nInstanceID				:= 131,
							sObjectName				:= OBJECT_NAME,
							sDescription			:= '{Benachrichtigung (Standard)}',
							eEventType				:= E_BA_EventType.eNotification,
							eAlarmMode				:= E_BA_AlarmMode.eStandard,
							aPriority				:= [ 133, 134, 135 ]
						);
	{endregion}
	{region 'Other'}
		OthSmpl			: FB_BA_EC := (
							iParent					:= THIS^,
							nInstanceID				:= 182,
							sObjectName				:= OBJECT_NAME,
							sDescription			:= '{Sonstiges (Einfach)}',
							eEventType				:= E_BA_EventType.eOther,
							eAlarmMode				:= E_BA_AlarmMode.eSimple,
							aPriority				:= [ 180, 181, 182 ]
						);
		OthStd			: FB_BA_EC := (
							iParent					:= THIS^,
							nInstanceID				:= 181,
							sObjectName				:= OBJECT_NAME,
							sDescription			:= '{Sonstiges (Standard)}',
							eEventType				:= E_BA_EventType.eOther,
							eAlarmMode				:= E_BA_AlarmMode.eStandard,
							aPriority				:= [ 183, 184, 185 ]
						);
	{endregion}
END_VAR

SUPER^(); // FB_BA_View
AlmSmpl(); // FB_BA_EC
AlmStd(); // FB_BA_EC
AlmExt(); // FB_BA_EC
DstSmpl(); // FB_BA_EC
DstStd(); // FB_BA_EC
DstExt(); // FB_BA_EC
MntnSmpl(); // FB_BA_EC
MntnStd(); // FB_BA_EC
MntnExt(); // FB_BA_EC
NtfSmpl(); // FB_BA_EC
NtfStd(); // FB_BA_EC
OthSmpl(); // FB_BA_EC
OthStd(); // FB_BA_EC

END_FUNCTION_BLOCK

// ---- SAMPLES/Demo/Supplement specific/BACnet/Optional Extensions/Events/FB_BACnet_MyLocalObjectEvents.TcPOU
FUNCTION_BLOCK FB_BACnet_MyLocalObjectEvents EXTENDS FB_BA_LocalObjectEventSubscriber

METHOD PROTECTED OnBACnetObjectStateChanged
VAR_INPUT
	iObject			: I_BA_Object;
	fbBACnetObject	: POINTER TO FB_BACnet_BaseObject;
	tState			: TCOM_STATE;
END_VAR
CASE (tState) OF
	TCOM_STATE.TCOM_STATE_PREOP:
		// Sample 1) Enable specific properties.
		CASE (fbBACnetObject^.ObjectType) OF
			E_BACnetObjType.ObjAnalogInput:
				// Sample 1.1) Enable 'PT1 damp factor' for all analog inputs:
				fbBACnetObject^.EnableProperty(E_BACnetPropIdentifier.PropPt1DampFactor, TRUE);
			
		END_CASE
		
		// Sample 2) Writeprotect specific properties.
		CASE (fbBACnetObject^.ObjectType) OF
			E_BACnetObjType.ObjSchedule:
				// Sample 2.1) Writeprotect 'schedule default' for all schedulers:
				fbBACnetObject^.WriteProtectProperty(E_BACnetPropIdentifier.PropScheduleDefault, TRUE);
			
		END_CASE
		
END_CASE
END_METHOD

METHOD PROTECTED OnInitStateChange
VAR_INPUT
	iObject			: I_BA_Object;
	eState			: E_BA_InitState;
END_VAR
VAR
	
	_fbBACnetObj	: POINTER TO FB_BACnet_BaseObject;
END_VAR
// Sample 1) Evaluate object state.
CASE (eState) OF
	E_BA_InitState.ePostInitSupplement:
		// Object has finished to initialize enabled supplement(s).
	
		// Sample 1.1) Initialize some properties:
		IF (iObject.IsReused) THEN
			; // Skip (Do not overwrite previously restored persisted values here).
		ELSIF (iObject.GetBACnetObject(fbObject=>_fbBACnetObj)) THEN
			CASE (_fbBACnetObj^.ObjectType) OF
				E_BACnetObjType.ObjAnalogInput:
					// Write 'PT1 damp factor' for all analog inputs:
					_fbBACnetObj^.WritePropertyReal(E_BACnetPropIdentifier.PropPt1DampFactor, 0.5);
				
			END_CASE
		END_IF

END_CASE
END_METHOD

END_FUNCTION_BLOCK

// ---- SAMPLES/Demo/[Helper]/FunctionBlocks/Nested/FB_SubSubNestedView.TcPOU
FUNCTION_BLOCK FB_SubSubNestedView EXTENDS FB_SubNestedView
VAR_INPUT CONSTANT
	SubX		: FB_SubNestedView		:= (iParent:=THIS^);
END_VAR

SUPER^();

SubX();

END_FUNCTION_BLOCK
